LIN {X 0,Y 720.208,Z 610.953,A -85,B 0,C 180,E1 34660.965,E2 34660.965} C_VEL
LIN {X 0,Y 720.172,Z 610.956,A -85,B 0,C 180,E1 34658.142,E2 34658.142} C_VEL
LIN {X 0,Y 720.181,Z 610.956,A -85,B 0,C 180,E1 34655.418,E2 34655.418} C_VEL
LIN {X 0,Y 720.141,Z 610.957,A -85,B 0,C 180,E1 34652.468,E2 34652.468} C_VEL
LIN {X 0,Y 720.162,Z 610.958,A -85,B 0,C 180,E1 34649.922,E2 34649.922} C_VEL
LIN {X 0,Y 720.219,Z 610.948,A -85,B 0,C 180,E1 34646.977,E2 34646.977} C_VEL
LIN {X 0,Y 720.22,Z 610.957,A -85,B 0,C 180,E1 34643.945,E2 34643.945} C_VEL
LIN {X 0,Y 720.198,Z 610.951,A -85,B 0,C 180,E1 34640.975,E2 34640.975} C_VEL
LIN {X 0,Y 720.16,Z 610.957,A -85,B 0,C 180,E1 34637.899,E2 34637.899} C_VEL
LIN {X 0,Y 720.131,Z 610.96,A -85,B 0,C 180,E1 34635.403,E2 34635.403} C_VEL
LIN {X 0,Y 720.218,Z 610.954,A -85,B 0,C 180,E1 34632.551,E2 34632.551} C_VEL
LIN {X 0,Y 720.177,Z 610.955,A -85,B 0,C 180,E1 34629.692,E2 34629.692} C_VEL
LIN {X 0,Y 720.205,Z 610.955,A -85,B 0,C 180,E1 34626.953,E2 34626.953} C_VEL
LIN {X 0,Y 720.215,Z 610.951,A -85,B 0,C 180,E1 34624.069,E2 34624.069} C_VEL
LIN {X 0,Y 720.163,Z 610.958,A -85,B 0,C 180,E1 34621.2,E2 34621.2} C_VEL
LIN {X 0,Y 720.152,Z 610.959,A -85,B 0,C 180,E1 34618.625,E2 34618.625} C_VEL
LIN {X 0,Y 720.156,Z 610.958,A -85,B 0,C 180,E1 34615.556,E2 34615.556} C_VEL
LIN {X 0,Y 720.173,Z 610.957,A -85,B 0,C 180,E1 34612.948,E2 34612.948} C_VEL
LIN {X 0,Y 720.219,Z 610.95,A -85,B 0,C 180,E1 34610.002,E2 34610.002} C_VEL
LIN {X 0,Y 720.219,Z 610.959,A -85,B 0,C 180,E1 34607.02,E2 34607.02} C_VEL
LIN {X 0,Y 720.18,Z 610.954,A -85,B 0,C 180,E1 34604.13,E2 34604.13} C_VEL
LIN {X 0,Y 720.174,Z 610.961,A -85,B 0,C 180,E1 34601.152,E2 34601.152} C_VEL
LIN {X 0,Y 720.13,Z 610.962,A -85,B 0,C 180,E1 34598.564,E2 34598.564} C_VEL
LIN {X 0,Y 720.234,Z 611.091,A -85,B 0,C 180,E1 34597.759,E2 34597.759} C_VEL
LIN {X 0,Y 721.518,Z 617.349,A -85,B 0,C 180,E1 34597.269,E2 34597.269} C_VEL
LIN {X 0,Y 721.444,Z 660.306,A -85,B 0,C 180,E1 34594.24,E2 34594.24} C_VEL
LIN {X 0,Y 721.342,Z 691.441,A -85,B 0,C 180,E1 34592.016,E2 34592.016} C_VEL
LIN {X 0,Y 721.105,Z 731.111,A -85,B 0,C 180,E1 34589.212,E2 34589.212} C_VEL
LIN {X 0,Y 720.893,Z 759.497,A -85,B 0,C 180,E1 34587.193,E2 34587.193} C_VEL
LIN {X 0,Y 720.617,Z 798.923,A -85,B 0,C 180,E1 34584.386,E2 34584.386} C_VEL
LIN {X 0,Y 720.526,Z 815.5,A -85,B 0,C 180,E1 34583.249,E2 34583.249} C_VEL
LIN {X 0,Y 720.895,Z 824.532,A -85,B 0,C 180,E1 34583.152,E2 34583.152} C_VEL
LIN {X 0,Y 720.697,Z 956.974,A -85,B 0,C 180,E1 34581.81,E2 34581.81} C_VEL
LIN {X 0,Y 720.607,Z 973.104,A -85,B 0,C 180,E1 34581.493,E2 34581.493} C_VEL
LIN {X 0,Y 720.51,Z 989.356,A -85,B 0,C 180,E1 34581.02,E2 34581.02} C_VEL
LIN {X 0,Y 720.374,Z 1004.011,A -85,B 0,C 180,E1 34580.429,E2 34580.429} C_VEL
LIN {X 0,Y 720.299,Z 1015.674,A -85,B 0,C 180,E1 34579.838,E2 34579.838} C_VEL
LIN {X 0,Y 720.212,Z 1026.341,A -85,B 0,C 180,E1 34579.184,E2 34579.184} C_VEL
LIN {X 0,Y 720.127,Z 1036.599,A -85,B 0,C 180,E1 34578.427,E2 34578.427} C_VEL
LIN {X 0,Y 720.06,Z 1045.774,A -85,B 0,C 180,E1 34577.619,E2 34577.619} C_VEL
LIN {X 0,Y 719.997,Z 1054.367,A -85,B 0,C 180,E1 34576.704,E2 34576.704} C_VEL
LIN {X 0,Y 719.964,Z 1062.582,A -85,B 0,C 180,E1 34575.628,E2 34575.628} C_VEL
LIN {X 0,Y 719.931,Z 1070.175,A -85,B 0,C 180,E1 34574.311,E2 34574.311} C_VEL
LIN {X 0,Y 719.92,Z 1074.932,A -85,B 0,C 180,E1 34573.164,E2 34573.164} C_VEL
LIN {X 0,Y 719.916,Z 1077.987,A -85,B 0,C 180,E1 34572.104,E2 34572.104} C_VEL
LIN {X 0,Y 719.915,Z 1079.89,A -85,B 0,C 180,E1 34570.967,E2 34570.967} C_VEL
LIN {X 0,Y 719.916,Z 1080.431,A -85,B 0,C 180,E1 34569.834,E2 34569.834} C_VEL
LIN {X 0,Y 719.915,Z 1079.432,A -85,B 0,C 180,E1 34568.545,E2 34568.545} C_VEL
LIN {X 0,Y 719.921,Z 1076.365,A -85,B 0,C 180,E1 34567.179,E2 34567.179} C_VEL
LIN {X 0,Y 719.925,Z 1071.892,A -85,B 0,C 180,E1 34565.977,E2 34565.977} C_VEL
LIN {X 0,Y 719.942,Z 1066.603,A -85,B 0,C 180,E1 34564.938,E2 34564.938} C_VEL
LIN {X 0,Y 719.967,Z 1060.414,A -85,B 0,C 180,E1 34563.98,E2 34563.98} C_VEL
LIN {X 0,Y 720.011,Z 1052.786,A -85,B 0,C 180,E1 34563.023,E2 34563.023} C_VEL
LIN {X 0,Y 720.083,Z 1043.455,A -85,B 0,C 180,E1 34562.067,E2 34562.067} C_VEL
LIN {X 0,Y 720.187,Z 1030.252,A -85,B 0,C 180,E1 34560.993,E2 34560.993} C_VEL
LIN {X 0,Y 720.28,Z 1018.57,A -85,B 0,C 180,E1 34560.237,E2 34560.237} C_VEL
LIN {X 0,Y 720.327,Z 1007.399,A -85,B 0,C 180,E1 34559.64,E2 34559.64} C_VEL
LIN {X 0,Y 720.427,Z 995.54,A -85,B 0,C 180,E1 34559.124,E2 34559.124} C_VEL
LIN {X 0,Y 720.552,Z 982.888,A -85,B 0,C 180,E1 34558.686,E2 34558.686} C_VEL
LIN {X 0,Y 720.627,Z 969.803,A -85,B 0,C 180,E1 34558.344,E2 34558.344} C_VEL
LIN {X 0,Y 720.709,Z 954.847,A -85,B 0,C 180,E1 34558.07,E2 34558.07} C_VEL
LIN {X 0,Y 720.676,Z 816.549,A -85,B 0,C 180,E1 34556.674,E2 34556.674} C_VEL
LIN {X 0,Y 720.51,Z 814.823,A -85,B 0,C 180,E1 34556.64,E2 34556.64} C_VEL
LIN {X 0,Y 720.829,Z 771.864,A -85,B 0,C 180,E1 34553.605,E2 34553.605} C_VEL
LIN {X 0,Y 721.072,Z 739.826,A -85,B 0,C 180,E1 34551.305,E2 34551.305} C_VEL
LIN {X 0,Y 721.215,Z 704.804,A -85,B 0,C 180,E1 34548.847,E2 34548.847} C_VEL
LIN {X 0,Y 721.206,Z 667.656,A -85,B 0,C 180,E1 34546.284,E2 34546.284} C_VEL
LIN {X 0,Y 721.014,Z 625.211,A -85,B 0,C 180,E1 34543.441,E2 34543.441} C_VEL
LIN {X 0,Y 720.81,Z 613.743,A -85,B 0,C 180,E1 34542.688,E2 34542.688} C_VEL
LIN {X 0,Y 720.216,Z 610.959,A -85,B 0,C 180,E1 34542.484,E2 34542.484} C_VEL
LIN {X 0,Y 720.181,Z 610.96,A -85,B 0,C 180,E1 34539.519,E2 34539.519} C_VEL
LIN {X 0,Y 720.186,Z 610.961,A -85,B 0,C 180,E1 34536.776,E2 34536.776} C_VEL
LIN {X 0,Y 720.22,Z 610.954,A -85,B 0,C 180,E1 34533.743,E2 34533.743} C_VEL
LIN {X 0,Y 720.175,Z 610.96,A -85,B 0,C 180,E1 34530.743,E2 34530.743} C_VEL
LIN {X 0,Y 720.19,Z 610.958,A -85,B 0,C 180,E1 34527.969,E2 34527.969} C_VEL
LIN {X 0,Y 720.208,Z 610.957,A -85,B 0,C 180,E1 34524.993,E2 34524.993} C_VEL
LIN {X 0,Y 720.195,Z 610.96,A -85,B 0,C 180,E1 34522.145,E2 34522.145} C_VEL
LIN {X 0,Y 720.222,Z 610.958,A -85,B 0,C 180,E1 34519.268,E2 34519.268} C_VEL
LIN {X 0,Y 720.216,Z 610.959,A -85,B 0,C 180,E1 34516.326,E2 34516.326} C_VEL
LIN {X 0,Y 720.223,Z 610.955,A -85,B 0,C 180,E1 34513.298,E2 34513.298} C_VEL
LIN {X 0,Y 720.175,Z 610.96,A -85,B 0,C 180,E1 34510.313,E2 34510.313} C_VEL
LIN {X 0,Y 720.196,Z 610.957,A -85,B 0,C 180,E1 34507.55,E2 34507.55} C_VEL
LIN {X 0,Y 720.195,Z 610.959,A -85,B 0,C 180,E1 34504.405,E2 34504.405} C_VEL
LIN {X 0,Y 720.21,Z 611.037,A -85,B 0,C 180,E1 34502.332,E2 34502.332} C_VEL
LIN {X 0,Y 723.137,Z 620.988,A -85,B 0,C 180,E1 34501.416,E2 34501.416} C_VEL
LIN {X 0,Y 722.601,Z 658.022,A -85,B 0,C 180,E1 34498.604,E2 34498.604} C_VEL
LIN {X 0,Y 722.325,Z 683.324,A -85,B 0,C 180,E1 34496.747,E2 34496.747} C_VEL
LIN {X 0,Y 723.83,Z 691.21,A -85,B 0,C 180,E1 34496.601,E2 34496.601} C_VEL
LIN {X 0,Y 723.03,Z 975.338,A -85,B 0,C 180,E1 34493.578,E2 34493.578} C_VEL
LIN {X 0,Y 722.886,Z 996.786,A -85,B 0,C 180,E1 34493.276,E2 34493.276} C_VEL
LIN {X 0,Y 722.659,Z 1019.236,A -85,B 0,C 180,E1 34492.811,E2 34492.811} C_VEL
LIN {X 0,Y 722.426,Z 1040.16,A -85,B 0,C 180,E1 34492.234,E2 34492.234} C_VEL
LIN {X 0,Y 722.134,Z 1060.43,A -85,B 0,C 180,E1 34491.525,E2 34491.525} C_VEL
LIN {X 0,Y 721.801,Z 1080.838,A -85,B 0,C 180,E1 34490.654,E2 34490.654} C_VEL
LIN {X 0,Y 721.49,Z 1100.586,A -85,B 0,C 180,E1 34489.646,E2 34489.646} C_VEL
LIN {X 0,Y 721.179,Z 1119.415,A -85,B 0,C 180,E1 34488.51,E2 34488.51} C_VEL
LIN {X 0,Y 720.868,Z 1136.909,A -85,B 0,C 180,E1 34487.266,E2 34487.266} C_VEL
LIN {X 0,Y 720.608,Z 1152.879,A -85,B 0,C 180,E1 34485.945,E2 34485.945} C_VEL
LIN {X 0,Y 720.414,Z 1167.469,A -85,B 0,C 180,E1 34484.548,E2 34484.548} C_VEL
LIN {X 0,Y 720.248,Z 1180.679,A -85,B 0,C 180,E1 34483.077,E2 34483.077} C_VEL
LIN {X 0,Y 720.109,Z 1192.4,A -85,B 0,C 180,E1 34481.533,E2 34481.533} C_VEL
LIN {X 0,Y 720.016,Z 1203.22,A -85,B 0,C 180,E1 34479.834,E2 34479.834} C_VEL
LIN {X 0,Y 719.975,Z 1211.702,A -85,B 0,C 180,E1 34478.223,E2 34478.223} C_VEL
LIN {X 0,Y 719.924,Z 1218.675,A -85,B 0,C 180,E1 34476.538,E2 34476.538} C_VEL
LIN {X 0,Y 719.904,Z 1224.199,A -85,B 0,C 180,E1 34474.779,E2 34474.779} C_VEL
LIN {X 0,Y 719.898,Z 1227.881,A -85,B 0,C 180,E1 34473.104,E2 34473.104} C_VEL
LIN {X 0,Y 719.898,Z 1229.883,A -85,B 0,C 180,E1 34471.431,E2 34471.431} C_VEL
LIN {X 0,Y 719.898,Z 1230.396,A -85,B 0,C 180,E1 34469.601,E2 34469.601} C_VEL
LIN {X 0,Y 719.915,Z 1229.336,A -85,B 0,C 180,E1 34467.929,E2 34467.929} C_VEL
LIN {X 0,Y 719.914,Z 1226.464,A -85,B 0,C 180,E1 34466.176,E2 34466.176} C_VEL
LIN {X 0,Y 719.917,Z 1221.903,A -85,B 0,C 180,E1 34464.42,E2 34464.42} C_VEL
LIN {X 0,Y 719.946,Z 1215.93,A -85,B 0,C 180,E1 34462.738,E2 34462.738} C_VEL
LIN {X 0,Y 719.984,Z 1208.468,A -85,B 0,C 180,E1 34461.131,E2 34461.131} C_VEL
LIN {X 0,Y 720.059,Z 1198.837,A -85,B 0,C 180,E1 34459.437,E2 34459.437} C_VEL
LIN {X 0,Y 720.162,Z 1188.342,A -85,B 0,C 180,E1 34457.897,E2 34457.897} C_VEL
LIN {X 0,Y 720.305,Z 1175.652,A -85,B 0,C 180,E1 34456.339,E2 34456.339} C_VEL
LIN {X 0,Y 720.484,Z 1161.703,A -85,B 0,C 180,E1 34454.875,E2 34454.875} C_VEL
LIN {X 0,Y 720.719,Z 1146.187,A -85,B 0,C 180,E1 34453.476,E2 34453.476} C_VEL
LIN {X 0,Y 721.006,Z 1129.487,A -85,B 0,C 180,E1 34452.18,E2 34452.18} C_VEL
LIN {X 0,Y 721.309,Z 1111.316,A -85,B 0,C 180,E1 34450.981,E2 34450.981} C_VEL
LIN {X 0,Y 721.617,Z 1092.115,A -85,B 0,C 180,E1 34449.901,E2 34449.901} C_VEL
LIN {X 0,Y 721.955,Z 1071.709,A -85,B 0,C 180,E1 34448.936,E2 34448.936} C_VEL
LIN {X 0,Y 722.287,Z 1051.348,A -85,B 0,C 180,E1 34448.136,E2 34448.136} C_VEL
LIN {X 0,Y 722.517,Z 1030.436,A -85,B 0,C 180,E1 34447.48,E2 34447.48} C_VEL
LIN {X 0,Y 722.782,Z 1007.95,A -85,B 0,C 180,E1 34446.936,E2 34446.936} C_VEL
LIN {X 0,Y 722.975,Z 986.397,A -85,B 0,C 180,E1 34446.559,E2 34446.559} C_VEL
LIN {X 0,Y 723.392,Z 834.871,A -85,B 0,C 180,E1 34444.934,E2 34444.934} C_VEL
LIN {X 0,Y 723.683,Z 689.443,A -85,B 0,C 180,E1 34443.374,E2 34443.374} C_VEL
LIN {X 0,Y 722.245,Z 682.748,A -85,B 0,C 180,E1 34443.235,E2 34443.235} C_VEL
LIN {X 0,Y 722.812,Z 644.848,A -85,B 0,C 180,E1 34440.405,E2 34440.405} C_VEL
LIN {X 0,Y 723.146,Z 620.604,A -85,B 0,C 180,E1 34438.554,E2 34438.554} C_VEL
LIN {X 0,Y 720.191,Z 610.959,A -85,B 0,C 180,E1 34437.664,E2 34437.664} C_VEL
LIN {X 0,Y 720.211,Z 610.953,A -85,B 0,C 180,E1 34434.819,E2 34434.819} C_VEL
LIN {X 0,Y 720.192,Z 610.958,A -85,B 0,C 180,E1 34431.842,E2 34431.842} C_VEL
LIN {X 0,Y 720.215,Z 610.949,A -85,B 0,C 180,E1 34428.927,E2 34428.927} C_VEL
LIN {X 0,Y 720.196,Z 610.959,A -85,B 0,C 180,E1 34425.873,E2 34425.873} C_VEL
LIN {X 0,Y 720.182,Z 610.953,A -85,B 0,C 180,E1 34423.086,E2 34423.086} C_VEL
LIN {X 0,Y 720.224,Z 610.959,A -85,B 0,C 180,E1 34420.096,E2 34420.096} C_VEL
LIN {X 0,Y 720.163,Z 610.956,A -85,B 0,C 180,E1 34417.291,E2 34417.291} C_VEL
LIN {X 0,Y 720.212,Z 610.953,A -85,B 0,C 180,E1 34414.503,E2 34414.503} C_VEL
LIN {X 0,Y 720.167,Z 610.961,A -85,B 0,C 180,E1 34411.516,E2 34411.516} C_VEL
LIN {X 0,Y 720.15,Z 610.961,A -85,B 0,C 180,E1 34408.985,E2 34408.985} C_VEL
LIN {X 0,Y 720.254,Z 611.202,A -85,B 0,C 180,E1 34407.94,E2 34407.94} C_VEL
LIN {X 0,Y 721.962,Z 619.154,A -85,B 0,C 180,E1 34407.153,E2 34407.153} C_VEL
LIN {X 0,Y 722.019,Z 624.53,A -85,B 0,C 180,E1 34406.701,E2 34406.701} C_VEL
LIN {X 0,Y 723.829,Z 632.779,A -85,B 0,C 180,E1 34406.539,E2 34406.539} C_VEL
LIN {X 0,Y 723.098,Z 895.124,A -85,B 0,C 180,E1 34403.747,E2 34403.747} C_VEL
LIN {X 0,Y 722.945,Z 929.462,A -85,B 0,C 180,E1 34403.351,E2 34403.351} C_VEL
LIN {X 0,Y 722.776,Z 950.86,A -85,B 0,C 180,E1 34402.96,E2 34402.96} C_VEL
LIN {X 0,Y 722.496,Z 972.696,A -85,B 0,C 180,E1 34402.411,E2 34402.411} C_VEL
LIN {X 0,Y 722.203,Z 994.686,A -85,B 0,C 180,E1 34401.696,E2 34401.696} C_VEL
LIN {X 0,Y 721.915,Z 1015.557,A -85,B 0,C 180,E1 34400.854,E2 34400.854} C_VEL
LIN {X 0,Y 721.574,Z 1035.207,A -85,B 0,C 180,E1 34399.894,E2 34399.894} C_VEL
LIN {X 0,Y 721.25,Z 1054.058,A -85,B 0,C 180,E1 34398.805,E2 34398.805} C_VEL
LIN {X 0,Y 720.952,Z 1072.496,A -85,B 0,C 180,E1 34397.554,E2 34397.554} C_VEL
LIN {X 0,Y 720.68,Z 1089.562,A -85,B 0,C 180,E1 34396.194,E2 34396.194} C_VEL
LIN {X 0,Y 720.453,Z 1104.64,A -85,B 0,C 180,E1 34394.797,E2 34394.797} C_VEL
LIN {X 0,Y 720.257,Z 1118.345,A -85,B 0,C 180,E1 34393.305,E2 34393.305} C_VEL
LIN {X 0,Y 720.127,Z 1130.91,A -85,B 0,C 180,E1 34391.698,E2 34391.698} C_VEL
LIN {X 0,Y 720.026,Z 1141.578,A -85,B 0,C 180,E1 34390.075,E2 34390.075} C_VEL
LIN {X 0,Y 719.964,Z 1150.276,A -85,B 0,C 180,E1 34388.467,E2 34388.467} C_VEL
LIN {X 0,Y 719.924,Z 1157.686,A -85,B 0,C 180,E1 34386.757,E2 34386.757} C_VEL
LIN {X 0,Y 719.917,Z 1163.454,A -85,B 0,C 180,E1 34385.021,E2 34385.021} C_VEL
LIN {X 0,Y 719.917,Z 1167.323,A -85,B 0,C 180,E1 34383.346,E2 34383.346} C_VEL
LIN {X 0,Y 719.914,Z 1169.711,A -85,B 0,C 180,E1 34381.593,E2 34381.593} C_VEL
LIN {X 0,Y 719.91,Z 1170.475,A -85,B 0,C 180,E1 34379.843,E2 34379.843} C_VEL
LIN {X 0,Y 719.911,Z 1169.52,A -85,B 0,C 180,E1 34378.092,E2 34378.092} C_VEL
LIN {X 0,Y 719.915,Z 1166.879,A -85,B 0,C 180,E1 34376.339,E2 34376.339} C_VEL
LIN {X 0,Y 719.926,Z 1162.567,A -85,B 0,C 180,E1 34374.583,E2 34374.583} C_VEL
LIN {X 0,Y 719.942,Z 1156.731,A -85,B 0,C 180,E1 34372.902,E2 34372.902} C_VEL
LIN {X 0,Y 719.976,Z 1149.125,A -85,B 0,C 180,E1 34371.215,E2 34371.215} C_VEL
LIN {X 0,Y 720.041,Z 1140.185,A -85,B 0,C 180,E1 34369.602,E2 34369.602} C_VEL
LIN {X 0,Y 720.135,Z 1129.841,A -85,B 0,C 180,E1 34368.062,E2 34368.062} C_VEL
LIN {X 0,Y 720.269,Z 1117.57,A -85,B 0,C 180,E1 34366.515,E2 34366.515} C_VEL
LIN {X 0,Y 720.461,Z 1103.912,A -85,B 0,C 180,E1 34365.042,E2 34365.042} C_VEL
LIN {X 0,Y 720.489,Z 1101.611,A -85,B 0,C 180,E1 34364.82,E2 34364.82} C_VEL
LIN {X 0,Y 719.582,Z 1096.843,A -85,B 0,C 180,E1 34364.341,E2 34364.341} C_VEL
LIN {X 0,Y 713.69,Z 1083.945,A -85,B 0,C 180,E1 34363.074,E2 34363.074} C_VEL
LIN {X 0,Y 713.042,Z 1079.38,A -85,B 0,C 180,E1 34362.686,E2 34362.686} C_VEL
LIN {X 0,Y 713.399,Z 1061.921,A -85,B 0,C 180,E1 34361.408,E2 34361.408} C_VEL
LIN {X 0,Y 713.782,Z 1043.036,A -85,B 0,C 180,E1 34360.229,E2 34360.229} C_VEL
LIN {X 0,Y 714.179,Z 1022.968,A -85,B 0,C 180,E1 34359.171,E2 34359.171} C_VEL
LIN {X 0,Y 714.582,Z 1002.755,A -85,B 0,C 180,E1 34358.28,E2 34358.28} C_VEL
LIN {X 0,Y 714.928,Z 981.908,A -85,B 0,C 180,E1 34357.534,E2 34357.534} C_VEL
LIN {X 0,Y 715.253,Z 959.699,A -85,B 0,C 180,E1 34356.905,E2 34356.905} C_VEL
LIN {X 0,Y 715.521,Z 937.487,A -85,B 0,C 180,E1 34356.436,E2 34356.436} C_VEL
LIN {X 0,Y 715.69,Z 915.823,A -85,B 0,C 180,E1 34356.126,E2 34356.126} C_VEL
LIN {X 0,Y 716.689,Z 640.954,A -85,B 0,C 180,E1 34353.175,E2 34353.175} C_VEL
LIN {X 0,Y 716.479,Z 632.558,A -85,B 0,C 180,E1 34353.074,E2 34353.074} C_VEL
LIN {X 0,Y 714.354,Z 623.95,A -85,B 0,C 180,E1 34352.878,E2 34352.878} C_VEL
LIN {X 0,Y 714.269,Z 619.697,A -85,B 0,C 180,E1 34352.489,E2 34352.489} C_VEL
LIN {X 0,Y 712.232,Z 611.949,A -85,B 0,C 180,E1 34351.671,E2 34351.671} C_VEL
LIN {X 0,Y 712.231,Z 611.95,A -85,B 0,C 180,E1 34348.99,E2 34348.99} C_VEL
LIN {X 0,Y 712.204,Z 611.949,A -85,B 0,C 180,E1 34345.935,E2 34345.935} C_VEL
LIN {X 0,Y 712.231,Z 611.948,A -85,B 0,C 180,E1 34343.373,E2 34343.373} C_VEL
LIN {X 0,Y 712.281,Z 611.938,A -85,B 0,C 180,E1 34340.411,E2 34340.411} C_VEL
LIN {X 0,Y 712.276,Z 611.948,A -85,B 0,C 180,E1 34337.358,E2 34337.358} C_VEL
LIN {X 0,Y 712.268,Z 611.94,A -85,B 0,C 180,E1 34334.355,E2 34334.355} C_VEL
LIN {X 0,Y 712.218,Z 611.949,A -85,B 0,C 180,E1 34331.395,E2 34331.395} C_VEL
LIN {X 0,Y 712.197,Z 611.949,A -85,B 0,C 180,E1 34328.871,E2 34328.871} C_VEL
LIN {X 0,Y 712.271,Z 611.942,A -85,B 0,C 180,E1 34325.909,E2 34325.909} C_VEL
LIN {X 0,Y 712.249,Z 611.946,A -85,B 0,C 180,E1 34323.004,E2 34323.004} C_VEL
LIN {X 0,Y 712.267,Z 611.939,A -85,B 0,C 180,E1 34320.078,E2 34320.078} C_VEL
LIN {X 0,Y 712.274,Z 611.948,A -85,B 0,C 180,E1 34317.055,E2 34317.055} C_VEL
LIN {X 0,Y 712.218,Z 611.946,A -85,B 0,C 180,E1 34314.29,E2 34314.29} C_VEL
LIN {X 0,Y 712.253,Z 611.949,A -85,B 0,C 180,E1 34311.408,E2 34311.408} C_VEL
LIN {X 0,Y 712.208,Z 611.946,A -85,B 0,C 180,E1 34308.67,E2 34308.67} C_VEL
LIN {X 0,Y 712.28,Z 611.946,A -85,B 0,C 180,E1 34305.888,E2 34305.888} C_VEL
LIN {X 0,Y 712.26,Z 611.939,A -85,B 0,C 180,E1 34302.981,E2 34302.981} C_VEL
LIN {X 0,Y 712.251,Z 611.944,A -85,B 0,C 180,E1 34300.108,E2 34300.108} C_VEL
LIN {X 0,Y 712.28,Z 611.94,A -85,B 0,C 180,E1 34297.178,E2 34297.178} C_VEL
LIN {X 0,Y 712.2,Z 611.948,A -85,B 0,C 180,E1 34294.349,E2 34294.349} C_VEL
LIN {X 0,Y 712.214,Z 611.946,A -85,B 0,C 180,E1 34291.743,E2 34291.743} C_VEL
LIN {X 0,Y 712.247,Z 611.942,A -85,B 0,C 180,E1 34288.634,E2 34288.634} C_VEL
LIN {X 0,Y 712.278,Z 611.945,A -85,B 0,C 180,E1 34285.734,E2 34285.734} C_VEL
LIN {X 0,Y 712.281,Z 611.938,A -85,B 0,C 180,E1 34282.743,E2 34282.743} C_VEL
LIN {X 0,Y 712.234,Z 611.944,A -85,B 0,C 180,E1 34279.758,E2 34279.758} C_VEL
LIN {X 0,Y 712.219,Z 611.945,A -85,B 0,C 180,E1 34277.103,E2 34277.103} C_VEL
LIN {X 0,Y 712.212,Z 611.947,A -85,B 0,C 180,E1 34274.029,E2 34274.029} C_VEL
LIN {X 0,Y 712.23,Z 611.946,A -85,B 0,C 180,E1 34271.418,E2 34271.418} C_VEL
LIN {X 0,Y 712.283,Z 611.938,A -85,B 0,C 180,E1 34268.422,E2 34268.422} C_VEL
LIN {X 0,Y 712.277,Z 611.948,A -85,B 0,C 180,E1 34265.361,E2 34265.361} C_VEL
LIN {X 0,Y 712.262,Z 611.941,A -85,B 0,C 180,E1 34262.404,E2 34262.404} C_VEL
LIN {X 0,Y 712.213,Z 611.948,A -85,B 0,C 180,E1 34259.379,E2 34259.379} C_VEL
LIN {X 0,Y 712.195,Z 611.949,A -85,B 0,C 180,E1 34256.899,E2 34256.899} C_VEL
LIN {X 0,Y 712.276,Z 611.942,A -85,B 0,C 180,E1 34253.953,E2 34253.953} C_VEL
LIN {X 0,Y 712.249,Z 611.946,A -85,B 0,C 180,E1 34251.031,E2 34251.031} C_VEL
LIN {X 0,Y 712.263,Z 611.941,A -85,B 0,C 180,E1 34248.181,E2 34248.181} C_VEL
LIN {X 0,Y 712.279,Z 611.947,A -85,B 0,C 180,E1 34245.143,E2 34245.143} C_VEL
LIN {X 0,Y 712.215,Z 611.947,A -85,B 0,C 180,E1 34242.364,E2 34242.364} C_VEL
LIN {X 0,Y 712.263,Z 611.949,A -85,B 0,C 180,E1 34239.486,E2 34239.486} C_VEL
LIN {X 0,Y 712.27,Z 612.124,A -85,B 0,C 180,E1 34237.952,E2 34237.952} C_VEL
LIN {X 0,Y 713.889,Z 619.31,A -85,B 0,C 180,E1 34237.387,E2 34237.387} C_VEL
LIN {X 0,Y 713.757,Z 663.317,A -85,B 0,C 180,E1 34234.26,E2 34234.26} C_VEL
LIN {X 0,Y 713.591,Z 701.946,A -85,B 0,C 180,E1 34231.507,E2 34231.507} C_VEL
LIN {X 0,Y 713.355,Z 742.215,A -85,B 0,C 180,E1 34228.642,E2 34228.642} C_VEL
LIN {X 0,Y 713.008,Z 777.238,A -85,B 0,C 180,E1 34226.123,E2 34226.123} C_VEL
LIN {X 0,Y 712.643,Z 815.347,A -85,B 0,C 180,E1 34223.401,E2 34223.401} C_VEL
LIN {X 0,Y 713.107,Z 823.548,A -85,B 0,C 180,E1 34223.309,E2 34223.309} C_VEL
LIN {X 0,Y 712.864,Z 956.883,A -85,B 0,C 180,E1 34221.943,E2 34221.943} C_VEL
LIN {X 0,Y 712.761,Z 972.125,A -85,B 0,C 180,E1 34221.643,E2 34221.643} C_VEL
LIN {X 0,Y 712.665,Z 987.139,A -85,B 0,C 180,E1 34221.22,E2 34221.22} C_VEL
LIN {X 0,Y 712.497,Z 1002.672,A -85,B 0,C 180,E1 34220.609,E2 34220.609} C_VEL
LIN {X 0,Y 712.392,Z 1015.074,A -85,B 0,C 180,E1 34219.982,E2 34219.982} C_VEL
LIN {X 0,Y 712.283,Z 1026.015,A -85,B 0,C 180,E1 34219.309,E2 34219.309} C_VEL
LIN {X 0,Y 712.183,Z 1035.86,A -85,B 0,C 180,E1 34218.582,E2 34218.582} C_VEL
LIN {X 0,Y 712.107,Z 1044.552,A -85,B 0,C 180,E1 34217.822,E2 34217.822} C_VEL
LIN {X 0,Y 712.035,Z 1052.626,A -85,B 0,C 180,E1 34216.981,E2 34216.981} C_VEL
LIN {X 0,Y 711.984,Z 1059.961,A -85,B 0,C 180,E1 34216.059,E2 34216.059} C_VEL
LIN {X 0,Y 711.951,Z 1065.949,A -85,B 0,C 180,E1 34215.141,E2 34215.141} C_VEL
LIN {X 0,Y 711.933,Z 1071.139,A -85,B 0,C 180,E1 34214.143,E2 34214.143} C_VEL
LIN {X 0,Y 711.92,Z 1075.087,A -85,B 0,C 180,E1 34213.15,E2 34213.15} C_VEL
LIN {X 0,Y 711.916,Z 1078.084,A -85,B 0,C 180,E1 34212.078,E2 34212.078} C_VEL
LIN {X 0,Y 711.916,Z 1079.881,A -85,B 0,C 180,E1 34210.974,E2 34210.974} C_VEL
LIN {X 0,Y 711.917,Z 1080.416,A -85,B 0,C 180,E1 34209.864,E2 34209.864} C_VEL
LIN {X 0,Y 711.915,Z 1079.531,A -85,B 0,C 180,E1 34208.608,E2 34208.608} C_VEL
LIN {X 0,Y 711.921,Z 1076.459,A -85,B 0,C 180,E1 34207.179,E2 34207.179} C_VEL
LIN {X 0,Y 711.928,Z 1072.379,A -85,B 0,C 180,E1 34206.045,E2 34206.045} C_VEL
LIN {X 0,Y 711.947,Z 1067.231,A -85,B 0,C 180,E1 34204.994,E2 34204.994} C_VEL
LIN {X 0,Y 711.976,Z 1061.192,A -85,B 0,C 180,E1 34204.025,E2 34204.025} C_VEL
LIN {X 0,Y 712.017,Z 1054.418,A -85,B 0,C 180,E1 34203.138,E2 34203.138} C_VEL
LIN {X 0,Y 712.088,Z 1046.234,A -85,B 0,C 180,E1 34202.251,E2 34202.251} C_VEL
LIN {X 0,Y 712.17,Z 1037.305,A -85,B 0,C 180,E1 34201.446,E2 34201.446} C_VEL
LIN {X 0,Y 712.264,Z 1027.776,A -85,B 0,C 180,E1 34200.722,E2 34200.722} C_VEL
LIN {X 0,Y 712.364,Z 1017.697,A -85,B 0,C 180,E1 34200.079,E2 34200.079} C_VEL
LIN {X 0,Y 712.429,Z 1007.182,A -85,B 0,C 180,E1 34199.516,E2 34199.516} C_VEL
LIN {X 0,Y 712.551,Z 995.271,A -85,B 0,C 180,E1 34198.993,E2 34198.993} C_VEL
LIN {X 0,Y 712.682,Z 983.862,A -85,B 0,C 180,E1 34198.591,E2 34198.591} C_VEL
LIN {X 0,Y 712.773,Z 971.223,A -85,B 0,C 180,E1 34198.247,E2 34198.247} C_VEL
LIN {X 0,Y 712.865,Z 956.628,A -85,B 0,C 180,E1 34197.964,E2 34197.964} C_VEL
LIN {X 0,Y 712.889,Z 817.239,A -85,B 0,C 180,E1 34196.533,E2 34196.533} C_VEL
LIN {X 0,Y 712.643,Z 814.973,A -85,B 0,C 180,E1 34196.499,E2 34196.499} C_VEL
LIN {X 0,Y 713.106,Z 772.038,A -85,B 0,C 180,E1 34193.396,E2 34193.396} C_VEL
LIN {X 0,Y 713.336,Z 745.498,A -85,B 0,C 180,E1 34191.494,E2 34191.494} C_VEL
LIN {X 0,Y 713.461,Z 706.642,A -85,B 0,C 180,E1 34188.765,E2 34188.765} C_VEL
LIN {X 0,Y 713.475,Z 670.947,A -85,B 0,C 180,E1 34186.298,E2 34186.298} C_VEL
LIN {X 0,Y 713.258,Z 630.642,A -85,B 0,C 180,E1 34183.591,E2 34183.591} C_VEL
LIN {X 0,Y 713.019,Z 615.291,A -85,B 0,C 180,E1 34182.577,E2 34182.577} C_VEL
LIN {X 0,Y 712.275,Z 611.947,A -85,B 0,C 180,E1 34182.326,E2 34182.326} C_VEL
LIN {X 0,Y 712.234,Z 611.949,A -85,B 0,C 180,E1 34179.28,E2 34179.28} C_VEL
LIN {X 0,Y 712.241,Z 611.95,A -85,B 0,C 180,E1 34176.59,E2 34176.59} C_VEL
LIN {X 0,Y 712.273,Z 611.945,A -85,B 0,C 180,E1 34173.485,E2 34173.485} C_VEL
LIN {X 0,Y 712.246,Z 611.949,A -85,B 0,C 180,E1 34170.569,E2 34170.569} C_VEL
LIN {X 0,Y 712.276,Z 611.946,A -85,B 0,C 180,E1 34167.665,E2 34167.665} C_VEL
LIN {X 0,Y 712.28,Z 611.948,A -85,B 0,C 180,E1 34164.644,E2 34164.644} C_VEL
LIN {X 0,Y 712.283,Z 611.944,A -85,B 0,C 180,E1 34161.562,E2 34161.562} C_VEL
LIN {X 0,Y 712.234,Z 611.948,A -85,B 0,C 180,E1 34158.498,E2 34158.498} C_VEL
LIN {X 0,Y 712.255,Z 611.946,A -85,B 0,C 180,E1 34155.719,E2 34155.719} C_VEL
LIN {X 0,Y 712.262,Z 611.945,A -85,B 0,C 180,E1 34152.641,E2 34152.641} C_VEL
LIN {X 0,Y 712.246,Z 611.949,A -85,B 0,C 180,E1 34149.801,E2 34149.801} C_VEL
LIN {X 0,Y 712.285,Z 611.946,A -85,B 0,C 180,E1 34146.826,E2 34146.826} C_VEL
LIN {X 0,Y 712.279,Z 611.949,A -85,B 0,C 180,E1 34143.868,E2 34143.868} C_VEL
LIN {X 0,Y 712.318,Z 612.184,A -85,B 0,C 180,E1 34142.623,E2 34142.623} C_VEL
LIN {X 0,Y 715.782,Z 623.742,A -85,B 0,C 180,E1 34141.556,E2 34141.556} C_VEL
LIN {X 0,Y 715.155,Z 660.411,A -85,B 0,C 180,E1 34138.746,E2 34138.746} C_VEL
LIN {X 0,Y 714.859,Z 683.329,A -85,B 0,C 180,E1 34137.049,E2 34137.049} C_VEL
LIN {X 0,Y 716.67,Z 692.713,A -85,B 0,C 180,E1 34136.872,E2 34136.872} C_VEL
LIN {X 0,Y 715.685,Z 976.194,A -85,B 0,C 180,E1 34133.824,E2 34133.824} C_VEL
LIN {X 0,Y 715.519,Z 997.499,A -85,B 0,C 180,E1 34133.518,E2 34133.518} C_VEL
LIN {X 0,Y 715.246,Z 1019.57,A -85,B 0,C 180,E1 34133.053,E2 34133.053} C_VEL
LIN {X 0,Y 714.973,Z 1039.924,A -85,B 0,C 180,E1 34132.486,E2 34132.486} C_VEL
LIN {X 0,Y 714.612,Z 1060.434,A -85,B 0,C 180,E1 34131.763,E2 34131.763} C_VEL
LIN {X 0,Y 714.215,Z 1081.097,A -85,B 0,C 180,E1 34130.871,E2 34130.871} C_VEL
LIN {X 0,Y 713.833,Z 1100.745,A -85,B 0,C 180,E1 34129.856,E2 34129.856} C_VEL
LIN {X 0,Y 713.454,Z 1119.415,A -85,B 0,C 180,E1 34128.718,E2 34128.718} C_VEL
LIN {X 0,Y 713.081,Z 1136.91,A -85,B 0,C 180,E1 34127.461,E2 34127.461} C_VEL
LIN {X 0,Y 712.772,Z 1152.879,A -85,B 0,C 180,E1 34126.125,E2 34126.125} C_VEL
LIN {X 0,Y 712.529,Z 1167.47,A -85,B 0,C 180,E1 34124.713,E2 34124.713} C_VEL
LIN {X 0,Y 712.319,Z 1180.678,A -85,B 0,C 180,E1 34123.225,E2 34123.225} C_VEL
LIN {X 0,Y 712.151,Z 1192.401,A -85,B 0,C 180,E1 34121.663,E2 34121.663} C_VEL
LIN {X 0,Y 712.042,Z 1203.22,A -85,B 0,C 180,E1 34119.945,E2 34119.945} C_VEL
LIN {X 0,Y 711.989,Z 1211.702,A -85,B 0,C 180,E1 34118.316,E2 34118.316} C_VEL
LIN {X 0,Y 711.926,Z 1218.675,A -85,B 0,C 180,E1 34116.612,E2 34116.612} C_VEL
LIN {X 0,Y 711.904,Z 1224.2,A -85,B 0,C 180,E1 34114.833,E2 34114.833} C_VEL
LIN {X 0,Y 711.9,Z 1227.881,A -85,B 0,C 180,E1 34113.139,E2 34113.139} C_VEL
LIN {X 0,Y 711.899,Z 1229.884,A -85,B 0,C 180,E1 34111.448,E2 34111.448} C_VEL
LIN {X 0,Y 711.898,Z 1230.396,A -85,B 0,C 180,E1 34109.597,E2 34109.597} C_VEL
LIN {X 0,Y 711.915,Z 1229.336,A -85,B 0,C 180,E1 34107.906,E2 34107.906} C_VEL
LIN {X 0,Y 711.915,Z 1226.463,A -85,B 0,C 180,E1 34106.133,E2 34106.133} C_VEL
LIN {X 0,Y 711.917,Z 1221.903,A -85,B 0,C 180,E1 34104.357,E2 34104.357} C_VEL
LIN {X 0,Y 711.95,Z 1215.93,A -85,B 0,C 180,E1 34102.656,E2 34102.656} C_VEL
LIN {X 0,Y 712,Z 1208.468,A -85,B 0,C 180,E1 34101.031,E2 34101.031} C_VEL
LIN {X 0,Y 712.086,Z 1198.836,A -85,B 0,C 180,E1 34099.317,E2 34099.317} C_VEL
LIN {X 0,Y 712.225,Z 1188.044,A -85,B 0,C 180,E1 34097.72,E2 34097.72} C_VEL
LIN {X 0,Y 712.393,Z 1175.739,A -85,B 0,C 180,E1 34096.195,E2 34096.195} C_VEL
LIN {X 0,Y 712.615,Z 1161.703,A -85,B 0,C 180,E1 34094.704,E2 34094.704} C_VEL
LIN {X 0,Y 712.891,Z 1146.683,A -85,B 0,C 180,E1 34093.33,E2 34093.33} C_VEL
LIN {X 0,Y 713.23,Z 1130.236,A -85,B 0,C 180,E1 34092.035,E2 34092.035} C_VEL
LIN {X 0,Y 713.582,Z 1112.76,A -85,B 0,C 180,E1 34090.859,E2 34090.859} C_VEL
LIN {X 0,Y 713.979,Z 1092.92,A -85,B 0,C 180,E1 34089.719,E2 34089.719} C_VEL
LIN {X 0,Y 714.378,Z 1073.484,A -85,B 0,C 180,E1 34088.778,E2 34088.778} C_VEL
LIN {X 0,Y 714.742,Z 1053.616,A -85,B 0,C 180,E1 34087.98,E2 34087.98} C_VEL
LIN {X 0,Y 715.049,Z 1032.653,A -85,B 0,C 180,E1 34087.297,E2 34087.297} C_VEL
LIN {X 0,Y 715.38,Z 1010.918,A -85,B 0,C 180,E1 34086.745,E2 34086.745} C_VEL
LIN {X 0,Y 715.577,Z 989.77,A -85,B 0,C 180,E1 34086.354,E2 34086.354} C_VEL
LIN {X 0,Y 715.772,Z 956.487,A -85,B 0,C 180,E1 34085.964,E2 34085.964} C_VEL
LIN {X 0,Y 716.63,Z 691.362,A -85,B 0,C 180,E1 34083.112,E2 34083.112} C_VEL
LIN {X 0,Y 714.779,Z 682.778,A -85,B 0,C 180,E1 34082.935,E2 34082.935} C_VEL
LIN {X 0,Y 715.458,Z 643.653,A -85,B 0,C 180,E1 34079.978,E2 34079.978} C_VEL
LIN {X 0,Y 715.71,Z 623.186,A -85,B 0,C 180,E1 34078.405,E2 34078.405} C_VEL
LIN {X 0,Y 712.259,Z 611.946,A -85,B 0,C 180,E1 34077.403,E2 34077.403} C_VEL
LIN {X 0,Y 712.271,Z 611.948,A -85,B 0,C 180,E1 34074.466,E2 34074.466} C_VEL
LIN {X 0,Y 712.244,Z 611.945,A -85,B 0,C 180,E1 34071.57,E2 34071.57} C_VEL
LIN {X 0,Y 712.277,Z 611.941,A -85,B 0,C 180,E1 34068.681,E2 34068.681} C_VEL
LIN {X 0,Y 712.245,Z 611.947,A -85,B 0,C 180,E1 34065.724,E2 34065.724} C_VEL
LIN {X 0,Y 712.261,Z 611.941,A -85,B 0,C 180,E1 34062.878,E2 34062.878} C_VEL
LIN {X 0,Y 712.252,Z 611.949,A -85,B 0,C 180,E1 34059.804,E2 34059.804} C_VEL
LIN {X 0,Y 712.227,Z 611.945,A -85,B 0,C 180,E1 34057.116,E2 34057.116} C_VEL
LIN {X 0,Y 712.282,Z 611.946,A -85,B 0,C 180,E1 34054.225,E2 34054.225} C_VEL
LIN {X 0,Y 712.22,Z 611.949,A -85,B 0,C 180,E1 34051.39,E2 34051.39} C_VEL
LIN {X 0,Y 712.222,Z 611.95,A -85,B 0,C 180,E1 34048.787,E2 34048.787} C_VEL
LIN {X 0,Y 712.285,Z 611.955,A -85,B 0,C 180,E1 34048.212,E2 34048.212} C_VEL
LIN {X 0,Y 714.389,Z 621.646,A -85,B 0,C 180,E1 34047.239,E2 34047.239} C_VEL
LIN {X 0,Y 714.465,Z 624.558,A -85,B 0,C 180,E1 34047.006,E2 34047.006} C_VEL
LIN {X 0,Y 716.665,Z 634.327,A -85,B 0,C 180,E1 34046.809,E2 34046.809} C_VEL
LIN {X 0,Y 715.771,Z 896.635,A -85,B 0,C 180,E1 34043.989,E2 34043.989} C_VEL
LIN {X 0,Y 715.591,Z 929.654,A -85,B 0,C 180,E1 34043.603,E2 34043.603} C_VEL
LIN {X 0,Y 715.386,Z 951.094,A -85,B 0,C 180,E1 34043.207,E2 34043.207} C_VEL
LIN {X 0,Y 715.059,Z 972.156,A -85,B 0,C 180,E1 34042.673,E2 34042.673} C_VEL
LIN {X 0,Y 714.735,Z 993.548,A -85,B 0,C 180,E1 34041.978,E2 34041.978} C_VEL
LIN {X 0,Y 714.38,Z 1013.672,A -85,B 0,C 180,E1 34041.17,E2 34041.17} C_VEL
LIN {X 0,Y 713.963,Z 1033.697,A -85,B 0,C 180,E1 34040.197,E2 34040.197} C_VEL
LIN {X 0,Y 713.571,Z 1053.411,A -85,B 0,C 180,E1 34039.057,E2 34039.057} C_VEL
LIN {X 0,Y 713.194,Z 1071.868,A -85,B 0,C 180,E1 34037.798,E2 34037.798} C_VEL
LIN {X 0,Y 712.868,Z 1088.615,A -85,B 0,C 180,E1 34036.461,E2 34036.461} C_VEL
LIN {X 0,Y 712.587,Z 1103.803,A -85,B 0,C 180,E1 34035.047,E2 34035.047} C_VEL
LIN {X 0,Y 712.356,Z 1117.475,A -85,B 0,C 180,E1 34033.558,E2 34033.558} C_VEL
LIN {X 0,Y 712.189,Z 1130.339,A -85,B 0,C 180,E1 34031.912,E2 34031.912} C_VEL
LIN {X 0,Y 712.061,Z 1141.089,A -85,B 0,C 180,E1 34030.274,E2 34030.274} C_VEL
LIN {X 0,Y 711.982,Z 1149.953,A -85,B 0,C 180,E1 34028.628,E2 34028.628} C_VEL
LIN {X 0,Y 711.931,Z 1157.599,A -85,B 0,C 180,E1 34026.858,E2 34026.858} C_VEL
LIN {X 0,Y 711.926,Z 1163.244,A -85,B 0,C 180,E1 34025.159,E2 34025.159} C_VEL
LIN {X 0,Y 711.917,Z 1167.168,A -85,B 0,C 180,E1 34023.464,E2 34023.464} C_VEL
LIN {X 0,Y 711.914,Z 1169.712,A -85,B 0,C 180,E1 34021.611,E2 34021.611} C_VEL
LIN {X 0,Y 711.91,Z 1170.475,A -85,B 0,C 180,E1 34019.841,E2 34019.841} C_VEL
LIN {X 0,Y 711.913,Z 1169.588,A -85,B 0,C 180,E1 34018.151,E2 34018.151} C_VEL
LIN {X 0,Y 711.916,Z 1167.037,A -85,B 0,C 180,E1 34016.378,E2 34016.378} C_VEL
LIN {X 0,Y 711.928,Z 1162.82,A -85,B 0,C 180,E1 34014.602,E2 34014.602} C_VEL
LIN {X 0,Y 711.947,Z 1157.036,A -85,B 0,C 180,E1 34012.903,E2 34012.903} C_VEL
LIN {X 0,Y 711.999,Z 1149.124,A -85,B 0,C 180,E1 34011.115,E2 34011.115} C_VEL
LIN {X 0,Y 712.077,Z 1140.184,A -85,B 0,C 180,E1 34009.484,E2 34009.484} C_VEL
LIN {X 0,Y 712.19,Z 1129.835,A -85,B 0,C 180,E1 34007.927,E2 34007.927} C_VEL
LIN {X 0,Y 712.372,Z 1116.863,A -85,B 0,C 180,E1 34006.28,E2 34006.28} C_VEL
LIN {X 0,Y 712.606,Z 1102.613,A -85,B 0,C 180,E1 34004.746,E2 34004.746} C_VEL
LIN {X 0,Y 712.888,Z 1087.247,A -85,B 0,C 180,E1 34003.33,E2 34003.33} C_VEL
LIN {X 0,Y 713.042,Z 1079.38,A -85,B 0,C 180,E1 34002.686,E2 34002.686} C_VEL
LIN {X 0,Y 712.178,Z 1074.006,A -85,B 0,C 180,E1 34002.24,E2 34002.24} C_VEL
LIN {X 0,Y 706.657,Z 1060.469,A -85,B 0,C 180,E1 34001.122,E2 34001.122} C_VEL
LIN {X 0,Y 705.853,Z 1054.615,A -85,B 0,C 180,E1 34000.713,E2 34000.713} C_VEL
LIN {X 0,Y 706.31,Z 1035.493,A -85,B 0,C 180,E1 33999.581,E2 33999.581} C_VEL
LIN {X 0,Y 706.785,Z 1015.703,A -85,B 0,C 180,E1 33998.595,E2 33998.595} C_VEL
LIN {X 0,Y 707.203,Z 995.552,A -85,B 0,C 180,E1 33997.762,E2 33997.762} C_VEL
LIN {X 0,Y 707.62,Z 973.57,A -85,B 0,C 180,E1 33997.026,E2 33997.026} C_VEL
LIN {X 0,Y 708.001,Z 951.788,A -85,B 0,C 180,E1 33996.461,E2 33996.461} C_VEL
LIN {X 0,Y 708.234,Z 930.159,A -85,B 0,C 180,E1 33996.055,E2 33996.055} C_VEL
LIN {X 0,Y 708.453,Z 898.268,A -85,B 0,C 180,E1 33995.674,E2 33995.674} C_VEL
LIN {X 0,Y 709.535,Z 634.886,A -85,B 0,C 180,E1 33992.815,E2 33992.815} C_VEL
LIN {X 0,Y 706.806,Z 623.919,A -85,B 0,C 180,E1 33992.562,E2 33992.562} C_VEL
LIN {X 0,Y 706.065,Z 619.69,A -85,B 0,C 180,E1 33992.142,E2 33992.142} C_VEL
LIN {X 0,Y 704.287,Z 612.938,A -85,B 0,C 180,E1 33991.419,E2 33991.419} C_VEL
LIN {X 0,Y 704.341,Z 612.938,A -85,B 0,C 180,E1 33988.508,E2 33988.508} C_VEL
LIN {X 0,Y 704.258,Z 612.939,A -85,B 0,C 180,E1 33985.694,E2 33985.694} C_VEL
LIN {X 0,Y 704.333,Z 612.937,A -85,B 0,C 180,E1 33982.995,E2 33982.995} C_VEL
LIN {X 0,Y 704.314,Z 612.93,A -85,B 0,C 180,E1 33979.979,E2 33979.979} C_VEL
LIN {X 0,Y 704.321,Z 612.934,A -85,B 0,C 180,E1 33977.1,E2 33977.1} C_VEL
LIN {X 0,Y 704.345,Z 612.929,A -85,B 0,C 180,E1 33974.189,E2 33974.189} C_VEL
LIN {X 0,Y 704.273,Z 612.937,A -85,B 0,C 180,E1 33971.314,E2 33971.314} C_VEL
LIN {X 0,Y 704.264,Z 612.938,A -85,B 0,C 180,E1 33968.765,E2 33968.765} C_VEL
LIN {X 0,Y 704.307,Z 612.931,A -85,B 0,C 180,E1 33965.697,E2 33965.697} C_VEL
LIN {X 0,Y 704.325,Z 612.936,A -85,B 0,C 180,E1 33962.82,E2 33962.82} C_VEL
LIN {X 0,Y 704.342,Z 612.926,A -85,B 0,C 180,E1 33959.793,E2 33959.793} C_VEL
LIN {X 0,Y 704.307,Z 612.934,A -85,B 0,C 180,E1 33956.747,E2 33956.747} C_VEL
LIN {X 0,Y 704.305,Z 612.934,A -85,B 0,C 180,E1 33953.956,E2 33953.956} C_VEL
LIN {X 0,Y 704.259,Z 612.938,A -85,B 0,C 180,E1 33950.907,E2 33950.907} C_VEL
LIN {X 0,Y 704.282,Z 612.936,A -85,B 0,C 180,E1 33948.373,E2 33948.373} C_VEL
LIN {X 0,Y 704.342,Z 612.927,A -85,B 0,C 180,E1 33945.396,E2 33945.396} C_VEL
LIN {X 0,Y 704.338,Z 612.935,A -85,B 0,C 180,E1 33942.379,E2 33942.379} C_VEL
LIN {X 0,Y 704.338,Z 612.927,A -85,B 0,C 180,E1 33939.314,E2 33939.314} C_VEL
LIN {X 0,Y 704.286,Z 612.937,A -85,B 0,C 180,E1 33936.359,E2 33936.359} C_VEL
LIN {X 0,Y 704.256,Z 612.937,A -85,B 0,C 180,E1 33933.827,E2 33933.827} C_VEL
LIN {X 0,Y 704.313,Z 612.933,A -85,B 0,C 180,E1 33930.815,E2 33930.815} C_VEL
LIN {X 0,Y 704.299,Z 612.934,A -85,B 0,C 180,E1 33928.035,E2 33928.035} C_VEL
LIN {X 0,Y 704.332,Z 612.927,A -85,B 0,C 180,E1 33925.115,E2 33925.115} C_VEL
LIN {X 0,Y 704.343,Z 612.936,A -85,B 0,C 180,E1 33922.086,E2 33922.086} C_VEL
LIN {X 0,Y 704.29,Z 612.93,A -85,B 0,C 180,E1 33919.231,E2 33919.231} C_VEL
LIN {X 0,Y 704.305,Z 612.937,A -85,B 0,C 180,E1 33916.287,E2 33916.287} C_VEL
LIN {X 0,Y 704.261,Z 612.936,A -85,B 0,C 180,E1 33913.59,E2 33913.59} C_VEL
LIN {X 0,Y 704.344,Z 612.933,A -85,B 0,C 180,E1 33910.772,E2 33910.772} C_VEL
LIN {X 0,Y 704.313,Z 612.932,A -85,B 0,C 180,E1 33907.815,E2 33907.815} C_VEL
LIN {X 0,Y 704.315,Z 612.932,A -85,B 0,C 180,E1 33904.974,E2 33904.974} C_VEL
LIN {X 0,Y 704.344,Z 612.932,A -85,B 0,C 180,E1 33902,E2 33902} C_VEL
LIN {X 0,Y 704.262,Z 612.937,A -85,B 0,C 180,E1 33899.169,E2 33899.169} C_VEL
LIN {X 0,Y 704.296,Z 612.938,A -85,B 0,C 180,E1 33896.48,E2 33896.48} C_VEL
LIN {X 0,Y 704.291,Z 612.933,A -85,B 0,C 180,E1 33893.466,E2 33893.466} C_VEL
LIN {X 0,Y 704.34,Z 612.937,A -85,B 0,C 180,E1 33890.614,E2 33890.614} C_VEL
LIN {X 0,Y 704.332,Z 612.929,A -85,B 0,C 180,E1 33887.575,E2 33887.575} C_VEL
LIN {X 0,Y 704.299,Z 612.935,A -85,B 0,C 180,E1 33884.644,E2 33884.644} C_VEL
LIN {X 0,Y 704.32,Z 612.935,A -85,B 0,C 180,E1 33881.816,E2 33881.816} C_VEL
LIN {X 0,Y 704.256,Z 612.941,A -85,B 0,C 180,E1 33878.866,E2 33878.866} C_VEL
LIN {X 0,Y 704.288,Z 613.003,A -85,B 0,C 180,E1 33878.163,E2 33878.163} C_VEL
LIN {X 0,Y 706.261,Z 621.413,A -85,B 0,C 180,E1 33877.498,E2 33877.498} C_VEL
LIN {X 0,Y 706.087,Z 666.858,A -85,B 0,C 180,E1 33874.254,E2 33874.254} C_VEL
LIN {X 0,Y 705.853,Z 707.108,A -85,B 0,C 180,E1 33871.369,E2 33871.369} C_VEL
LIN {X 0,Y 705.574,Z 747.48,A -85,B 0,C 180,E1 33868.478,E2 33868.478} C_VEL
LIN {X 0,Y 705.205,Z 782.039,A -85,B 0,C 180,E1 33865.982,E2 33865.982} C_VEL
LIN {X 0,Y 704.848,Z 815.904,A -85,B 0,C 180,E1 33863.548,E2 33863.548} C_VEL
LIN {X 0,Y 705.319,Z 824.238,A -85,B 0,C 180,E1 33863.451,E2 33863.451} C_VEL
LIN {X 0,Y 705.03,Z 957.286,A -85,B 0,C 180,E1 33862.07,E2 33862.07} C_VEL
LIN {X 0,Y 704.92,Z 972.372,A -85,B 0,C 180,E1 33861.77,E2 33861.77} C_VEL
LIN {X 0,Y 704.807,Z 987.54,A -85,B 0,C 180,E1 33861.337,E2 33861.337} C_VEL
LIN {X 0,Y 704.617,Z 1002.557,A -85,B 0,C 180,E1 33860.737,E2 33860.737} C_VEL
LIN {X 0,Y 704.479,Z 1015.213,A -85,B 0,C 180,E1 33860.087,E2 33860.087} C_VEL
LIN {X 0,Y 704.357,Z 1025.694,A -85,B 0,C 180,E1 33859.436,E2 33859.436} C_VEL
LIN {X 0,Y 704.242,Z 1035.445,A -85,B 0,C 180,E1 33858.714,E2 33858.714} C_VEL
LIN {X 0,Y 704.147,Z 1044.219,A -85,B 0,C 180,E1 33857.943,E2 33857.943} C_VEL
LIN {X 0,Y 704.063,Z 1052.331,A -85,B 0,C 180,E1 33857.094,E2 33857.094} C_VEL
LIN {X 0,Y 703.999,Z 1059.717,A -85,B 0,C 180,E1 33856.161,E2 33856.161} C_VEL
LIN {X 0,Y 703.962,Z 1065.75,A -85,B 0,C 180,E1 33855.232,E2 33855.232} C_VEL
LIN {X 0,Y 703.935,Z 1070.981,A -85,B 0,C 180,E1 33854.223,E2 33854.223} C_VEL
LIN {X 0,Y 703.924,Z 1074.968,A -85,B 0,C 180,E1 33853.218,E2 33853.218} C_VEL
LIN {X 0,Y 703.918,Z 1077.82,A -85,B 0,C 180,E1 33852.217,E2 33852.217} C_VEL
LIN {X 0,Y 703.916,Z 1079.703,A -85,B 0,C 180,E1 33851.137,E2 33851.137} C_VEL
LIN {X 0,Y 703.917,Z 1080.399,A -85,B 0,C 180,E1 33850.06,E2 33850.06} C_VEL
LIN {X 0,Y 703.917,Z 1079.932,A -85,B 0,C 180,E1 33848.987,E2 33848.987} C_VEL
LIN {X 0,Y 703.917,Z 1078.305,A -85,B 0,C 180,E1 33847.918,E2 33847.918} C_VEL
LIN {X 0,Y 703.92,Z 1075.48,A -85,B 0,C 180,E1 33846.849,E2 33846.849} C_VEL
LIN {X 0,Y 703.929,Z 1071.784,A -85,B 0,C 180,E1 33845.868,E2 33845.868} C_VEL
LIN {X 0,Y 703.952,Z 1066.937,A -85,B 0,C 180,E1 33844.887,E2 33844.887} C_VEL
LIN {X 0,Y 703.987,Z 1061.401,A -85,B 0,C 180,E1 33843.989,E2 33843.989} C_VEL
LIN {X 0,Y 704.037,Z 1054.671,A -85,B 0,C 180,E1 33843.092,E2 33843.092} C_VEL
LIN {X 0,Y 704.118,Z 1046.538,A -85,B 0,C 180,E1 33842.196,E2 33842.196} C_VEL
LIN {X 0,Y 704.207,Z 1038.657,A -85,B 0,C 180,E1 33841.463,E2 33841.463} C_VEL
LIN {X 0,Y 704.319,Z 1028.79,A -85,B 0,C 180,E1 33840.69,E2 33840.69} C_VEL
LIN {X 0,Y 704.441,Z 1018.213,A -85,B 0,C 180,E1 33839.998,E2 33839.998} C_VEL
LIN {X 0,Y 704.53,Z 1007.868,A -85,B 0,C 180,E1 33839.429,E2 33839.429} C_VEL
LIN {X 0,Y 704.675,Z 996.166,A -85,B 0,C 180,E1 33838.901,E2 33838.901} C_VEL
LIN {X 0,Y 704.822,Z 984.966,A -85,B 0,C 180,E1 33838.494,E2 33838.494} C_VEL
LIN {X 0,Y 704.93,Z 972.176,A -85,B 0,C 180,E1 33838.136,E2 33838.136} C_VEL
LIN {X 0,Y 705.029,Z 957.568,A -85,B 0,C 180,E1 33837.844,E2 33837.844} C_VEL
LIN {X 0,Y 705.21,Z 861.519,A -85,B 0,C 180,E1 33836.841,E2 33836.841} C_VEL
LIN {X 0,Y 705.09,Z 817.797,A -85,B 0,C 180,E1 33836.387,E2 33836.387} C_VEL
LIN {X 0,Y 704.894,Z 815.689,A -85,B 0,C 180,E1 33836.339,E2 33836.339} C_VEL
LIN {X 0,Y 705.356,Z 775.226,A -85,B 0,C 180,E1 33833.405,E2 33833.405} C_VEL
LIN {X 0,Y 705.575,Z 739.025,A -85,B 0,C 180,E1 33830.825,E2 33830.825} C_VEL
LIN {X 0,Y 705.748,Z 703.823,A -85,B 0,C 180,E1 33828.351,E2 33828.351} C_VEL
LIN {X 0,Y 705.71,Z 666.95,A -85,B 0,C 180,E1 33825.81,E2 33825.81} C_VEL
LIN {X 0,Y 705.524,Z 622.066,A -85,B 0,C 180,E1 33822.811,E2 33822.811} C_VEL
LIN {X 0,Y 705.245,Z 616.915,A -85,B 0,C 180,E1 33822.464,E2 33822.464} C_VEL
LIN {X 0,Y 704.34,Z 612.935,A -85,B 0,C 180,E1 33822.185,E2 33822.185} C_VEL
LIN {X 0,Y 704.297,Z 612.938,A -85,B 0,C 180,E1 33819.088,E2 33819.088} C_VEL
LIN {X 0,Y 704.301,Z 612.939,A -85,B 0,C 180,E1 33816.398,E2 33816.398} C_VEL
LIN {X 0,Y 704.334,Z 612.935,A -85,B 0,C 180,E1 33813.345,E2 33813.345} C_VEL
LIN {X 0,Y 704.324,Z 612.938,A -85,B 0,C 180,E1 33810.392,E2 33810.392} C_VEL
LIN {X 0,Y 704.342,Z 612.937,A -85,B 0,C 180,E1 33807.449,E2 33807.449} C_VEL
LIN {X 0,Y 704.328,Z 612.937,A -85,B 0,C 180,E1 33804.504,E2 33804.504} C_VEL
LIN {X 0,Y 704.344,Z 612.932,A -85,B 0,C 180,E1 33801.448,E2 33801.448} C_VEL
LIN {X 0,Y 704.295,Z 612.937,A -85,B 0,C 180,E1 33798.43,E2 33798.43} C_VEL
LIN {X 0,Y 704.321,Z 612.935,A -85,B 0,C 180,E1 33795.566,E2 33795.566} C_VEL
LIN {X 0,Y 704.327,Z 612.935,A -85,B 0,C 180,E1 33792.51,E2 33792.51} C_VEL
LIN {X 0,Y 704.331,Z 612.938,A -85,B 0,C 180,E1 33789.568,E2 33789.568} C_VEL
LIN {X 0,Y 704.334,Z 612.938,A -85,B 0,C 180,E1 33786.599,E2 33786.599} C_VEL
LIN {X 0,Y 704.331,Z 612.938,A -85,B 0,C 180,E1 33783.704,E2 33783.704} C_VEL
LIN {X 0,Y 704.356,Z 613.042,A -85,B 0,C 180,E1 33782.947,E2 33782.947} C_VEL
LIN {X 0,Y 708.384,Z 626.81,A -85,B 0,C 180,E1 33781.663,E2 33781.663} C_VEL
LIN {X 0,Y 707.727,Z 662.203,A -85,B 0,C 180,E1 33778.938,E2 33778.938} C_VEL
LIN {X 0,Y 707.405,Z 683.292,A -85,B 0,C 180,E1 33777.358,E2 33777.358} C_VEL
LIN {X 0,Y 709.526,Z 694.112,A -85,B 0,C 180,E1 33777.149,E2 33777.149} C_VEL
LIN {X 0,Y 708.357,Z 976.73,A -85,B 0,C 180,E1 33774.079,E2 33774.079} C_VEL
LIN {X 0,Y 708.167,Z 998.018,A -85,B 0,C 180,E1 33773.768,E2 33773.768} C_VEL
LIN {X 0,Y 707.845,Z 1019.873,A -85,B 0,C 180,E1 33773.3,E2 33773.3} C_VEL
LIN {X 0,Y 707.497,Z 1041.206,A -85,B 0,C 180,E1 33772.693,E2 33772.693} C_VEL
LIN {X 0,Y 707.088,Z 1061.669,A -85,B 0,C 180,E1 33771.958,E2 33771.958} C_VEL
LIN {X 0,Y 706.648,Z 1081.093,A -85,B 0,C 180,E1 33771.105,E2 33771.105} C_VEL
LIN {X 0,Y 706.19,Z 1100.741,A -85,B 0,C 180,E1 33770.08,E2 33770.08} C_VEL
LIN {X 0,Y 705.737,Z 1119.415,A -85,B 0,C 180,E1 33768.931,E2 33768.931} C_VEL
LIN {X 0,Y 705.309,Z 1136.911,A -85,B 0,C 180,E1 33767.659,E2 33767.659} C_VEL
LIN {X 0,Y 704.943,Z 1152.878,A -85,B 0,C 180,E1 33766.309,E2 33766.309} C_VEL
LIN {X 0,Y 704.649,Z 1167.471,A -85,B 0,C 180,E1 33764.881,E2 33764.881} C_VEL
LIN {X 0,Y 704.394,Z 1180.676,A -85,B 0,C 180,E1 33763.377,E2 33763.377} C_VEL
LIN {X 0,Y 704.198,Z 1192.399,A -85,B 0,C 180,E1 33761.797,E2 33761.797} C_VEL
LIN {X 0,Y 704.067,Z 1203.221,A -85,B 0,C 180,E1 33760.059,E2 33760.059} C_VEL
LIN {X 0,Y 704.001,Z 1211.703,A -85,B 0,C 180,E1 33758.411,E2 33758.411} C_VEL
LIN {X 0,Y 703.931,Z 1218.676,A -85,B 0,C 180,E1 33756.688,E2 33756.688} C_VEL
LIN {X 0,Y 703.905,Z 1224.2,A -85,B 0,C 180,E1 33754.888,E2 33754.888} C_VEL
LIN {X 0,Y 703.9,Z 1227.881,A -85,B 0,C 180,E1 33753.175,E2 33753.175} C_VEL
LIN {X 0,Y 703.899,Z 1229.884,A -85,B 0,C 180,E1 33751.464,E2 33751.464} C_VEL
LIN {X 0,Y 703.898,Z 1230.396,A -85,B 0,C 180,E1 33749.592,E2 33749.592} C_VEL
LIN {X 0,Y 703.914,Z 1229.23,A -85,B 0,C 180,E1 33747.801,E2 33747.801} C_VEL
LIN {X 0,Y 703.918,Z 1226.303,A -85,B 0,C 180,E1 33746.008,E2 33746.008} C_VEL
LIN {X 0,Y 703.918,Z 1221.65,A -85,B 0,C 180,E1 33744.211,E2 33744.211} C_VEL
LIN {X 0,Y 703.953,Z 1215.58,A -85,B 0,C 180,E1 33742.49,E2 33742.49} C_VEL
LIN {X 0,Y 704.017,Z 1208.062,A -85,B 0,C 180,E1 33740.846,E2 33740.846} C_VEL
LIN {X 0,Y 704.119,Z 1198.321,A -85,B 0,C 180,E1 33739.112,E2 33739.112} C_VEL
LIN {X 0,Y 704.286,Z 1187.718,A -85,B 0,C 180,E1 33737.537,E2 33737.537} C_VEL
LIN {X 0,Y 704.496,Z 1175.035,A -85,B 0,C 180,E1 33735.953,E2 33735.953} C_VEL
LIN {X 0,Y 704.754,Z 1161.703,A -85,B 0,C 180,E1 33734.529,E2 33734.529} C_VEL
LIN {X 0,Y 705.09,Z 1146.187,A -85,B 0,C 180,E1 33733.099,E2 33733.099} C_VEL
LIN {X 0,Y 705.49,Z 1129.676,A -85,B 0,C 180,E1 33731.788,E2 33731.788} C_VEL
LIN {X 0,Y 705.905,Z 1112.512,A -85,B 0,C 180,E1 33730.626,E2 33730.626} C_VEL
LIN {X 0,Y 706.371,Z 1092.922,A -85,B 0,C 180,E1 33729.491,E2 33729.491} C_VEL
LIN {X 0,Y 706.829,Z 1073.392,A -85,B 0,C 180,E1 33728.536,E2 33728.536} C_VEL
LIN {X 0,Y 707.26,Z 1053.613,A -85,B 0,C 180,E1 33727.735,E2 33727.735} C_VEL
LIN {X 0,Y 707.622,Z 1032.65,A -85,B 0,C 180,E1 33727.045,E2 33727.045} C_VEL
LIN {X 0,Y 708.004,Z 1010.92,A -85,B 0,C 180,E1 33726.489,E2 33726.489} C_VEL
LIN {X 0,Y 708.243,Z 989.77,A -85,B 0,C 180,E1 33726.094,E2 33726.094} C_VEL
LIN {X 0,Y 708.464,Z 956.42,A -85,B 0,C 180,E1 33725.699,E2 33725.699} C_VEL
LIN {X 0,Y 709.482,Z 692.744,A -85,B 0,C 180,E1 33722.834,E2 33722.834} C_VEL
LIN {X 0,Y 707.334,Z 682.778,A -85,B 0,C 180,E1 33722.627,E2 33722.627} C_VEL
LIN {X 0,Y 708.095,Z 644.233,A -85,B 0,C 180,E1 33719.68,E2 33719.68} C_VEL
LIN {X 0,Y 708.12,Z 625.43,A -85,B 0,C 180,E1 33718.265,E2 33718.265} C_VEL
LIN {X 0,Y 704.339,Z 612.933,A -85,B 0,C 180,E1 33717.135,E2 33717.135} C_VEL
LIN {X 0,Y 704.326,Z 612.938,A -85,B 0,C 180,E1 33714.003,E2 33714.003} C_VEL
LIN {X 0,Y 704.333,Z 612.929,A -85,B 0,C 180,E1 33711.031,E2 33711.031} C_VEL
LIN {X 0,Y 704.324,Z 612.938,A -85,B 0,C 180,E1 33707.927,E2 33707.927} C_VEL
LIN {X 0,Y 704.317,Z 612.93,A -85,B 0,C 180,E1 33704.992,E2 33704.992} C_VEL
LIN {X 0,Y 704.32,Z 612.938,A -85,B 0,C 180,E1 33701.855,E2 33701.855} C_VEL
LIN {X 0,Y 704.295,Z 612.933,A -85,B 0,C 180,E1 33699.051,E2 33699.051} C_VEL
LIN {X 0,Y 704.344,Z 612.936,A -85,B 0,C 180,E1 33696.097,E2 33696.097} C_VEL
LIN {X 0,Y 704.28,Z 612.937,A -85,B 0,C 180,E1 33693.232,E2 33693.232} C_VEL
LIN {X 0,Y 704.329,Z 612.934,A -85,B 0,C 180,E1 33690.453,E2 33690.453} C_VEL
LIN {X 0,Y 704.318,Z 612.956,A -85,B 0,C 180,E1 33688.468,E2 33688.468} C_VEL
LIN {X 0,Y 706.819,Z 623.895,A -85,B 0,C 180,E1 33687.349,E2 33687.349} C_VEL
LIN {X 0,Y 709.519,Z 635.778,A -85,B 0,C 180,E1 33687.085,E2 33687.085} C_VEL
LIN {X 0,Y 708.455,Z 898.815,A -85,B 0,C 180,E1 33684.23,E2 33684.23} C_VEL
LIN {X 0,Y 708.244,Z 930.275,A -85,B 0,C 180,E1 33683.853,E2 33683.853} C_VEL
LIN {X 0,Y 708.005,Z 952.055,A -85,B 0,C 180,E1 33683.443,E2 33683.443} C_VEL
LIN {X 0,Y 707.613,Z 973.649,A -85,B 0,C 180,E1 33682.882,E2 33682.882} C_VEL
LIN {X 0,Y 707.219,Z 994.945,A -85,B 0,C 180,E1 33682.171,E2 33682.171} C_VEL
LIN {X 0,Y 706.811,Z 1014.651,A -85,B 0,C 180,E1 33681.364,E2 33681.364} C_VEL
LIN {X 0,Y 706.33,Z 1034.517,A -85,B 0,C 180,E1 33680.381,E2 33680.381} C_VEL
LIN {X 0,Y 705.872,Z 1053.927,A -85,B 0,C 180,E1 33679.241,E2 33679.241} C_VEL
LIN {X 0,Y 705.432,Z 1071.949,A -85,B 0,C 180,E1 33677.994,E2 33677.994} C_VEL
LIN {X 0,Y 705.042,Z 1088.617,A -85,B 0,C 180,E1 33676.649,E2 33676.649} C_VEL
LIN {X 0,Y 704.717,Z 1103.812,A -85,B 0,C 180,E1 33675.219,E2 33675.219} C_VEL
LIN {X 0,Y 704.453,Z 1117.482,A -85,B 0,C 180,E1 33673.713,E2 33673.713} C_VEL
LIN {X 0,Y 704.246,Z 1130.34,A -85,B 0,C 180,E1 33672.048,E2 33672.048} C_VEL
LIN {X 0,Y 704.096,Z 1141.09,A -85,B 0,C 180,E1 33670.392,E2 33670.392} C_VEL
LIN {X 0,Y 704,Z 1149.878,A -85,B 0,C 180,E1 33668.743,E2 33668.743} C_VEL
LIN {X 0,Y 703.941,Z 1157.602,A -85,B 0,C 180,E1 33666.936,E2 33666.936} C_VEL
LIN {X 0,Y 703.931,Z 1163.243,A -85,B 0,C 180,E1 33665.217,E2 33665.217} C_VEL
LIN {X 0,Y 703.918,Z 1167.17,A -85,B 0,C 180,E1 33663.503,E2 33663.503} C_VEL
LIN {X 0,Y 703.914,Z 1169.713,A -85,B 0,C 180,E1 33661.63,E2 33661.63} C_VEL
LIN {X 0,Y 703.91,Z 1170.475,A -85,B 0,C 180,E1 33659.839,E2 33659.839} C_VEL
LIN {X 0,Y 703.912,Z 1169.586,A -85,B 0,C 180,E1 33658.13,E2 33658.13} C_VEL
LIN {X 0,Y 703.915,Z 1167.037,A -85,B 0,C 180,E1 33656.337,E2 33656.337} C_VEL
LIN {X 0,Y 703.929,Z 1162.82,A -85,B 0,C 180,E1 33654.541,E2 33654.541} C_VEL
LIN {X 0,Y 703.956,Z 1157.032,A -85,B 0,C 180,E1 33652.822,E2 33652.822} C_VEL
LIN {X 0,Y 704.016,Z 1149.123,A -85,B 0,C 180,E1 33651.014,E2 33651.014} C_VEL
LIN {X 0,Y 704.112,Z 1139.937,A -85,B 0,C 180,E1 33649.324,E2 33649.324} C_VEL
LIN {X 0,Y 704.26,Z 1129.243,A -85,B 0,C 180,E1 33647.706,E2 33647.706} C_VEL
LIN {X 0,Y 704.467,Z 1116.861,A -85,B 0,C 180,E1 33646.123,E2 33646.123} C_VEL
LIN {X 0,Y 704.733,Z 1103.059,A -85,B 0,C 180,E1 33644.616,E2 33644.616} C_VEL
LIN {X 0,Y 705.071,Z 1087.288,A -85,B 0,C 180,E1 33643.144,E2 33643.144} C_VEL
LIN {X 0,Y 705.47,Z 1070.277,A -85,B 0,C 180,E1 33641.791,E2 33641.791} C_VEL
LIN {X 0,Y 705.853,Z 1054.615,A -85,B 0,C 180,E1 33640.713,E2 33640.713} C_VEL
LIN {X 0,Y 705.065,Z 1048.697,A -85,B 0,C 180,E1 33640.313,E2 33640.313} C_VEL
LIN {X 0,Y 699.546,Z 1032.974,A -85,B 0,C 180,E1 33639.237,E2 33639.237} C_VEL
LIN {X 0,Y 698.921,Z 1027.536,A -85,B 0,C 180,E1 33638.928,E2 33638.928} C_VEL
LIN {X 0,Y 699.433,Z 1007.819,A -85,B 0,C 180,E1 33638.006,E2 33638.006} C_VEL
LIN {X 0,Y 699.916,Z 987.709,A -85,B 0,C 180,E1 33637.225,E2 33637.225} C_VEL
LIN {X 0,Y 700.386,Z 966.328,A -85,B 0,C 180,E1 33636.56,E2 33636.56} C_VEL
LIN {X 0,Y 700.712,Z 944.697,A -85,B 0,C 180,E1 33636.051,E2 33636.051} C_VEL
LIN {X 0,Y 701.01,Z 921.94,A -85,B 0,C 180,E1 33635.675,E2 33635.675} C_VEL
LIN {X 0,Y 702.395,Z 645.496,A -85,B 0,C 180,E1 33632.636,E2 33632.636} C_VEL
LIN {X 0,Y 702.219,Z 635.693,A -85,B 0,C 180,E1 33632.518,E2 33632.518} C_VEL
LIN {X 0,Y 699.025,Z 624.07,A -85,B 0,C 180,E1 33632.245,E2 33632.245} C_VEL
LIN {X 0,Y 696.357,Z 613.926,A -85,B 0,C 180,E1 33631.151,E2 33631.151} C_VEL
LIN {X 0,Y 696.341,Z 613.93,A -85,B 0,C 180,E1 33628.063,E2 33628.063} C_VEL
LIN {X 0,Y 696.332,Z 613.928,A -85,B 0,C 180,E1 33625.366,E2 33625.366} C_VEL
LIN {X 0,Y 696.397,Z 613.918,A -85,B 0,C 180,E1 33622.398,E2 33622.398} C_VEL
LIN {X 0,Y 696.389,Z 613.924,A -85,B 0,C 180,E1 33619.425,E2 33619.425} C_VEL
LIN {X 0,Y 696.401,Z 613.916,A -85,B 0,C 180,E1 33616.325,E2 33616.325} C_VEL
LIN {X 0,Y 696.355,Z 613.925,A -85,B 0,C 180,E1 33613.285,E2 33613.285} C_VEL
LIN {X 0,Y 696.333,Z 613.926,A -85,B 0,C 180,E1 33610.687,E2 33610.687} C_VEL
LIN {X 0,Y 696.336,Z 613.925,A -85,B 0,C 180,E1 33607.506,E2 33607.506} C_VEL
LIN {X 0,Y 696.361,Z 613.924,A -85,B 0,C 180,E1 33604.854,E2 33604.854} C_VEL
LIN {X 0,Y 696.399,Z 613.916,A -85,B 0,C 180,E1 33601.794,E2 33601.794} C_VEL
LIN {X 0,Y 696.389,Z 613.925,A -85,B 0,C 180,E1 33598.751,E2 33598.751} C_VEL
LIN {X 0,Y 696.395,Z 613.918,A -85,B 0,C 180,E1 33595.789,E2 33595.789} C_VEL
LIN {X 0,Y 696.326,Z 613.925,A -85,B 0,C 180,E1 33592.805,E2 33592.805} C_VEL
LIN {X 0,Y 696.33,Z 613.927,A -85,B 0,C 180,E1 33590.247,E2 33590.247} C_VEL
LIN {X 0,Y 696.364,Z 613.92,A -85,B 0,C 180,E1 33587.12,E2 33587.12} C_VEL
LIN {X 0,Y 696.402,Z 613.924,A -85,B 0,C 180,E1 33584.214,E2 33584.214} C_VEL
LIN {X 0,Y 696.4,Z 613.917,A -85,B 0,C 180,E1 33581.177,E2 33581.177} C_VEL
LIN {X 0,Y 696.363,Z 613.922,A -85,B 0,C 180,E1 33578.256,E2 33578.256} C_VEL
LIN {X 0,Y 696.353,Z 613.924,A -85,B 0,C 180,E1 33575.522,E2 33575.522} C_VEL
LIN {X 0,Y 696.325,Z 613.923,A -85,B 0,C 180,E1 33572.47,E2 33572.47} C_VEL
LIN {X 0,Y 696.353,Z 613.925,A -85,B 0,C 180,E1 33569.837,E2 33569.837} C_VEL
LIN {X 0,Y 696.394,Z 613.914,A -85,B 0,C 180,E1 33566.791,E2 33566.791} C_VEL
LIN {X 0,Y 696.393,Z 613.924,A -85,B 0,C 180,E1 33563.737,E2 33563.737} C_VEL
LIN {X 0,Y 696.401,Z 613.917,A -85,B 0,C 180,E1 33560.747,E2 33560.747} C_VEL
LIN {X 0,Y 696.338,Z 613.923,A -85,B 0,C 180,E1 33557.816,E2 33557.816} C_VEL
LIN {X 0,Y 696.321,Z 613.927,A -85,B 0,C 180,E1 33555.277,E2 33555.277} C_VEL
LIN {X 0,Y 696.364,Z 613.921,A -85,B 0,C 180,E1 33552.193,E2 33552.193} C_VEL
LIN {X 0,Y 696.384,Z 613.924,A -85,B 0,C 180,E1 33549.318,E2 33549.318} C_VEL
LIN {X 0,Y 696.398,Z 613.916,A -85,B 0,C 180,E1 33546.207,E2 33546.207} C_VEL
LIN {X 0,Y 696.369,Z 613.924,A -85,B 0,C 180,E1 33543.203,E2 33543.203} C_VEL
LIN {X 0,Y 696.373,Z 613.922,A -85,B 0,C 180,E1 33540.402,E2 33540.402} C_VEL
LIN {X 0,Y 696.323,Z 613.927,A -85,B 0,C 180,E1 33537.421,E2 33537.421} C_VEL
LIN {X 0,Y 696.342,Z 613.926,A -85,B 0,C 180,E1 33534.846,E2 33534.846} C_VEL
LIN {X 0,Y 696.388,Z 613.918,A -85,B 0,C 180,E1 33531.771,E2 33531.771} C_VEL
LIN {X 0,Y 696.403,Z 613.925,A -85,B 0,C 180,E1 33528.777,E2 33528.777} C_VEL
LIN {X 0,Y 696.404,Z 613.917,A -85,B 0,C 180,E1 33525.752,E2 33525.752} C_VEL
LIN {X 0,Y 696.346,Z 613.927,A -85,B 0,C 180,E1 33522.776,E2 33522.776} C_VEL
LIN {X 0,Y 696.325,Z 613.929,A -85,B 0,C 180,E1 33520.191,E2 33520.191} C_VEL
LIN {X 0,Y 696.341,Z 614.058,A -85,B 0,C 180,E1 33518.362,E2 33518.362} C_VEL
LIN {X 0,Y 698.619,Z 623.346,A -85,B 0,C 180,E1 33517.617,E2 33517.617} C_VEL
LIN {X 0,Y 698.421,Z 666.95,A -85,B 0,C 180,E1 33514.494,E2 33514.494} C_VEL
LIN {X 0,Y 698.157,Z 706.998,A -85,B 0,C 180,E1 33511.61,E2 33511.61} C_VEL
LIN {X 0,Y 697.833,Z 746.898,A -85,B 0,C 180,E1 33508.733,E2 33508.733} C_VEL
LIN {X 0,Y 697.433,Z 783.557,A -85,B 0,C 180,E1 33506.08,E2 33506.08} C_VEL
LIN {X 0,Y 697.094,Z 816.81,A -85,B 0,C 180,E1 33503.693,E2 33503.693} C_VEL
LIN {X 0,Y 697.539,Z 825.005,A -85,B 0,C 180,E1 33503.597,E2 33503.597} C_VEL
LIN {X 0,Y 697.195,Z 958.266,A -85,B 0,C 180,E1 33502.19,E2 33502.19} C_VEL
LIN {X 0,Y 697.085,Z 974.09,A -85,B 0,C 180,E1 33501.87,E2 33501.87} C_VEL
LIN {X 0,Y 696.94,Z 990.698,A -85,B 0,C 180,E1 33501.369,E2 33501.369} C_VEL
LIN {X 0,Y 696.761,Z 1004.099,A -85,B 0,C 180,E1 33500.813,E2 33500.813} C_VEL
LIN {X 0,Y 696.617,Z 1016.406,A -85,B 0,C 180,E1 33500.168,E2 33500.168} C_VEL
LIN {X 0,Y 696.47,Z 1026.94,A -85,B 0,C 180,E1 33499.497,E2 33499.497} C_VEL
LIN {X 0,Y 696.329,Z 1036.586,A -85,B 0,C 180,E1 33498.761,E2 33498.761} C_VEL
LIN {X 0,Y 696.212,Z 1045.146,A -85,B 0,C 180,E1 33497.983,E2 33497.983} C_VEL
LIN {X 0,Y 696.105,Z 1053.091,A -85,B 0,C 180,E1 33497.123,E2 33497.123} C_VEL
LIN {X 0,Y 696.03,Z 1059.708,A -85,B 0,C 180,E1 33496.266,E2 33496.266} C_VEL
LIN {X 0,Y 695.975,Z 1065.681,A -85,B 0,C 180,E1 33495.326,E2 33495.326} C_VEL
LIN {X 0,Y 695.939,Z 1070.849,A -85,B 0,C 180,E1 33494.305,E2 33494.305} C_VEL
LIN {X 0,Y 695.926,Z 1074.848,A -85,B 0,C 180,E1 33493.288,E2 33493.288} C_VEL
LIN {X 0,Y 695.919,Z 1077.737,A -85,B 0,C 180,E1 33492.275,E2 33492.275} C_VEL
LIN {X 0,Y 695.916,Z 1079.655,A -85,B 0,C 180,E1 33491.182,E2 33491.182} C_VEL
LIN {X 0,Y 695.916,Z 1080.385,A -85,B 0,C 180,E1 33490.093,E2 33490.093} C_VEL
LIN {X 0,Y 695.917,Z 1079.952,A -85,B 0,C 180,E1 33489.008,E2 33489.008} C_VEL
LIN {X 0,Y 695.918,Z 1078.359,A -85,B 0,C 180,E1 33487.926,E2 33487.926} C_VEL
LIN {X 0,Y 695.922,Z 1075.71,A -85,B 0,C 180,E1 33486.888,E2 33486.888} C_VEL
LIN {X 0,Y 695.932,Z 1071.926,A -85,B 0,C 180,E1 33485.853,E2 33485.853} C_VEL
LIN {X 0,Y 695.962,Z 1067.224,A -85,B 0,C 180,E1 33484.861,E2 33484.861} C_VEL
LIN {X 0,Y 696.015,Z 1061.28,A -85,B 0,C 180,E1 33483.87,E2 33483.87} C_VEL
LIN {X 0,Y 696.088,Z 1054.593,A -85,B 0,C 180,E1 33482.962,E2 33482.962} C_VEL
LIN {X 0,Y 696.186,Z 1047.309,A -85,B 0,C 180,E1 33482.138,E2 33482.138} C_VEL
LIN {X 0,Y 696.311,Z 1038.623,A -85,B 0,C 180,E1 33481.315,E2 33481.315} C_VEL
LIN {X 0,Y 696.456,Z 1028.733,A -85,B 0,C 180,E1 33480.533,E2 33480.533} C_VEL
LIN {X 0,Y 696.598,Z 1018.086,A -85,B 0,C 180,E1 33479.834,E2 33479.834} C_VEL
LIN {X 0,Y 696.715,Z 1006.693,A -85,B 0,C 180,E1 33479.217,E2 33479.217} C_VEL
LIN {X 0,Y 696.897,Z 993.431,A -85,B 0,C 180,E1 33478.642,E2 33478.642} C_VEL
LIN {X 0,Y 697.086,Z 976.17,A -85,B 0,C 180,E1 33478.092,E2 33478.092} C_VEL
LIN {X 0,Y 697.191,Z 959.879,A -85,B 0,C 180,E1 33477.746,E2 33477.746} C_VEL
LIN {X 0,Y 697.276,Z 921.867,A -85,B 0,C 180,E1 33477.323,E2 33477.323} C_VEL
LIN {X 0,Y 697.333,Z 818.64,A -85,B 0,C 180,E1 33476.242,E2 33476.242} C_VEL
LIN {X 0,Y 697.164,Z 817.1,A -85,B 0,C 180,E1 33476.216,E2 33476.216} C_VEL
LIN {X 0,Y 697.628,Z 773.781,A -85,B 0,C 180,E1 33473.083,E2 33473.083} C_VEL
LIN {X 0,Y 697.861,Z 737.186,A -85,B 0,C 180,E1 33470.473,E2 33470.473} C_VEL
LIN {X 0,Y 698.087,Z 699.213,A -85,B 0,C 180,E1 33467.802,E2 33467.802} C_VEL
LIN {X 0,Y 697.919,Z 659.126,A -85,B 0,C 180,E1 33465.054,E2 33465.054} C_VEL
LIN {X 0,Y 697.75,Z 619.782,A -85,B 0,C 180,E1 33462.442,E2 33462.442} C_VEL
LIN {X 0,Y 696.404,Z 613.923,A -85,B 0,C 180,E1 33461.996,E2 33461.996} C_VEL
LIN {X 0,Y 696.364,Z 613.927,A -85,B 0,C 180,E1 33458.952,E2 33458.952} C_VEL
LIN {X 0,Y 696.377,Z 613.928,A -85,B 0,C 180,E1 33456.113,E2 33456.113} C_VEL
LIN {X 0,Y 696.4,Z 613.926,A -85,B 0,C 180,E1 33453.109,E2 33453.109} C_VEL
LIN {X 0,Y 696.405,Z 613.925,A -85,B 0,C 180,E1 33450.116,E2 33450.116} C_VEL
LIN {X 0,Y 696.37,Z 613.926,A -85,B 0,C 180,E1 33447.127,E2 33447.127} C_VEL
LIN {X 0,Y 696.378,Z 613.925,A -85,B 0,C 180,E1 33444.34,E2 33444.34} C_VEL
LIN {X 0,Y 696.395,Z 613.922,A -85,B 0,C 180,E1 33441.225,E2 33441.225} C_VEL
LIN {X 0,Y 696.359,Z 613.926,A -85,B 0,C 180,E1 33438.299,E2 33438.299} C_VEL
LIN {X 0,Y 696.402,Z 613.923,A -85,B 0,C 180,E1 33435.287,E2 33435.287} C_VEL
LIN {X 0,Y 696.399,Z 613.924,A -85,B 0,C 180,E1 33432.216,E2 33432.216} C_VEL
LIN {X 0,Y 696.408,Z 613.922,A -85,B 0,C 180,E1 33429.164,E2 33429.164} C_VEL
LIN {X 0,Y 696.361,Z 613.928,A -85,B 0,C 180,E1 33426.165,E2 33426.165} C_VEL
LIN {X 0,Y 696.395,Z 613.989,A -85,B 0,C 180,E1 33423.273,E2 33423.273} C_VEL
LIN {X 0,Y 701.01,Z 628.866,A -85,B 0,C 180,E1 33421.852,E2 33421.852} C_VEL
LIN {X 0,Y 700.276,Z 665.19,A -85,B 0,C 180,E1 33419.041,E2 33419.041} C_VEL
LIN {X 0,Y 699.978,Z 683.286,A -85,B 0,C 180,E1 33417.673,E2 33417.673} C_VEL
LIN {X 0,Y 702.4,Z 695.47,A -85,B 0,C 180,E1 33417.432,E2 33417.432} C_VEL
LIN {X 0,Y 701.042,Z 977.459,A -85,B 0,C 180,E1 33414.337,E2 33414.337} C_VEL
LIN {X 0,Y 700.824,Z 998.991,A -85,B 0,C 180,E1 33414.016,E2 33414.016} C_VEL
LIN {X 0,Y 700.452,Z 1020.638,A -85,B 0,C 180,E1 33413.541,E2 33413.541} C_VEL
LIN {X 0,Y 700.03,Z 1042.489,A -85,B 0,C 180,E1 33412.905,E2 33412.905} C_VEL
LIN {X 0,Y 699.57,Z 1063.072,A -85,B 0,C 180,E1 33412.151,E2 33412.151} C_VEL
LIN {X 0,Y 699.031,Z 1083.186,A -85,B 0,C 180,E1 33411.244,E2 33411.244} C_VEL
LIN {X 0,Y 698.495,Z 1102.941,A -85,B 0,C 180,E1 33410.18,E2 33410.18} C_VEL
LIN {X 0,Y 697.974,Z 1121.466,A -85,B 0,C 180,E1 33409.003,E2 33409.003} C_VEL
LIN {X 0,Y 697.501,Z 1138.628,A -85,B 0,C 180,E1 33407.729,E2 33407.729} C_VEL
LIN {X 0,Y 697.096,Z 1153.804,A -85,B 0,C 180,E1 33406.412,E2 33406.412} C_VEL
LIN {X 0,Y 696.735,Z 1169.022,A -85,B 0,C 180,E1 33404.884,E2 33404.884} C_VEL
LIN {X 0,Y 696.453,Z 1182,A -85,B 0,C 180,E1 33403.363,E2 33403.363} C_VEL
LIN {X 0,Y 696.234,Z 1193.544,A -85,B 0,C 180,E1 33401.766,E2 33401.766} C_VEL
LIN {X 0,Y 696.089,Z 1203.682,A -85,B 0,C 180,E1 33400.092,E2 33400.092} C_VEL
LIN {X 0,Y 696.008,Z 1212.41,A -85,B 0,C 180,E1 33398.342,E2 33398.342} C_VEL
LIN {X 0,Y 695.935,Z 1218.978,A -85,B 0,C 180,E1 33396.682,E2 33396.682} C_VEL
LIN {X 0,Y 695.908,Z 1224.2,A -85,B 0,C 180,E1 33394.944,E2 33394.944} C_VEL
LIN {X 0,Y 695.901,Z 1227.881,A -85,B 0,C 180,E1 33393.211,E2 33393.211} C_VEL
LIN {X 0,Y 695.9,Z 1229.884,A -85,B 0,C 180,E1 33391.481,E2 33391.481} C_VEL
LIN {X 0,Y 695.899,Z 1230.396,A -85,B 0,C 180,E1 33389.587,E2 33389.587} C_VEL
LIN {X 0,Y 695.914,Z 1229.231,A -85,B 0,C 180,E1 33387.776,E2 33387.776} C_VEL
LIN {X 0,Y 695.92,Z 1226.302,A -85,B 0,C 180,E1 33385.962,E2 33385.962} C_VEL
LIN {X 0,Y 695.922,Z 1221.651,A -85,B 0,C 180,E1 33384.144,E2 33384.144} C_VEL
LIN {X 0,Y 695.961,Z 1215.58,A -85,B 0,C 180,E1 33382.404,E2 33382.404} C_VEL
LIN {X 0,Y 696.035,Z 1207.977,A -85,B 0,C 180,E1 33380.723,E2 33380.723} C_VEL
LIN {X 0,Y 696.157,Z 1198.32,A -85,B 0,C 180,E1 33378.986,E2 33378.986} C_VEL
LIN {X 0,Y 696.347,Z 1187.717,A -85,B 0,C 180,E1 33377.392,E2 33377.392} C_VEL
LIN {X 0,Y 696.595,Z 1175.036,A -85,B 0,C 180,E1 33375.79,E2 33375.79} C_VEL
LIN {X 0,Y 696.91,Z 1161.268,A -85,B 0,C 180,E1 33374.307,E2 33374.307} C_VEL
LIN {X 0,Y 697.309,Z 1145.684,A -85,B 0,C 180,E1 33372.862,E2 33372.862} C_VEL
LIN {X 0,Y 697.763,Z 1129.09,A -85,B 0,C 180,E1 33371.536,E2 33371.536} C_VEL
LIN {X 0,Y 698.261,Z 1111.417,A -85,B 0,C 180,E1 33370.335,E2 33370.335} C_VEL
LIN {X 0,Y 698.769,Z 1093.043,A -85,B 0,C 180,E1 33369.264,E2 33369.264} C_VEL
LIN {X 0,Y 699.284,Z 1073.809,A -85,B 0,C 180,E1 33368.311,E2 33368.311} C_VEL
LIN {X 0,Y 699.791,Z 1053.609,A -85,B 0,C 180,E1 33367.484,E2 33367.484} C_VEL
LIN {X 0,Y 700.214,Z 1032.648,A -85,B 0,C 180,E1 33366.788,E2 33366.788} C_VEL
LIN {X 0,Y 700.643,Z 1010.922,A -85,B 0,C 180,E1 33366.226,E2 33366.226} C_VEL
LIN {X 0,Y 700.927,Z 989.607,A -85,B 0,C 180,E1 33365.826,E2 33365.826} C_VEL
LIN {X 0,Y 701.177,Z 955.366,A -85,B 0,C 180,E1 33365.419,E2 33365.419} C_VEL
LIN {X 0,Y 702.368,Z 694.229,A -85,B 0,C 180,E1 33362.553,E2 33362.553} C_VEL
LIN {X 0,Y 699.915,Z 682.539,A -85,B 0,C 180,E1 33362.293,E2 33362.293} C_VEL
LIN {X 0,Y 700.514,Z 650.266,A -85,B 0,C 180,E1 33359.838,E2 33359.838} C_VEL
LIN {X 0,Y 700.55,Z 627.785,A -85,B 0,C 180,E1 33358.13,E2 33358.13} C_VEL
LIN {X 0,Y 696.396,Z 613.925,A -85,B 0,C 180,E1 33356.86,E2 33356.86} C_VEL
LIN {X 0,Y 696.377,Z 613.927,A -85,B 0,C 180,E1 33353.833,E2 33353.833} C_VEL
LIN {X 0,Y 696.402,Z 613.918,A -85,B 0,C 180,E1 33350.836,E2 33350.836} C_VEL
LIN {X 0,Y 696.373,Z 613.926,A -85,B 0,C 180,E1 33347.779,E2 33347.779} C_VEL
LIN {X 0,Y 696.394,Z 613.918,A -85,B 0,C 180,E1 33344.822,E2 33344.822} C_VEL
LIN {X 0,Y 696.373,Z 613.927,A -85,B 0,C 180,E1 33341.778,E2 33341.778} C_VEL
LIN {X 0,Y 696.362,Z 613.922,A -85,B 0,C 180,E1 33338.971,E2 33338.971} C_VEL
LIN {X 0,Y 696.393,Z 613.927,A -85,B 0,C 180,E1 33335.923,E2 33335.923} C_VEL
LIN {X 0,Y 696.341,Z 613.926,A -85,B 0,C 180,E1 33333.16,E2 33333.16} C_VEL
LIN {X 0,Y 696.409,Z 613.924,A -85,B 0,C 180,E1 33330.264,E2 33330.264} C_VEL
LIN {X 0,Y 696.348,Z 613.945,A -85,B 0,C 180,E1 33328.754,E2 33328.754} C_VEL
LIN {X 0,Y 699.097,Z 624.487,A -85,B 0,C 180,E1 33327.652,E2 33327.652} C_VEL
LIN {X 0,Y 702.393,Z 636.465,A -85,B 0,C 180,E1 33327.376,E2 33327.376} C_VEL
LIN {X 0,Y 701.158,Z 899.503,A -85,B 0,C 180,E1 33324.491,E2 33324.491} C_VEL
LIN {X 0,Y 700.922,Z 930.386,A -85,B 0,C 180,E1 33324.116,E2 33324.116} C_VEL
LIN {X 0,Y 700.641,Z 952.218,A -85,B 0,C 180,E1 33323.702,E2 33323.702} C_VEL
LIN {X 0,Y 700.218,Z 972.793,A -85,B 0,C 180,E1 33323.164,E2 33323.164} C_VEL
LIN {X 0,Y 699.754,Z 994.708,A -85,B 0,C 180,E1 33322.429,E2 33322.429} C_VEL
LIN {X 0,Y 699.268,Z 1014.656,A -85,B 0,C 180,E1 33321.606,E2 33321.606} C_VEL
LIN {X 0,Y 698.728,Z 1034.534,A -85,B 0,C 180,E1 33320.613,E2 33320.613} C_VEL
LIN {X 0,Y 698.188,Z 1054.101,A -85,B 0,C 180,E1 33319.45,E2 33319.45} C_VEL
LIN {X 0,Y 697.667,Z 1072.539,A -85,B 0,C 180,E1 33318.157,E2 33318.157} C_VEL
LIN {X 0,Y 697.204,Z 1089.567,A -85,B 0,C 180,E1 33316.755,E2 33316.755} C_VEL
LIN {X 0,Y 696.837,Z 1104.653,A -85,B 0,C 180,E1 33315.31,E2 33315.31} C_VEL
LIN {X 0,Y 696.533,Z 1118.195,A -85,B 0,C 180,E1 33313.788,E2 33313.788} C_VEL
LIN {X 0,Y 696.294,Z 1130.926,A -85,B 0,C 180,E1 33312.104,E2 33312.104} C_VEL
LIN {X 0,Y 696.121,Z 1141.558,A -85,B 0,C 180,E1 33310.429,E2 33310.429} C_VEL
LIN {X 0,Y 696.014,Z 1150.289,A -85,B 0,C 180,E1 33308.761,E2 33308.761} C_VEL
LIN {X 0,Y 695.952,Z 1157.606,A -85,B 0,C 180,E1 33307.016,E2 33307.016} C_VEL
LIN {X 0,Y 695.93,Z 1163.453,A -85,B 0,C 180,E1 33305.195,E2 33305.195} C_VEL
LIN {X 0,Y 695.918,Z 1167.329,A -85,B 0,C 180,E1 33303.461,E2 33303.461} C_VEL
LIN {X 0,Y 695.914,Z 1169.713,A -85,B 0,C 180,E1 33301.648,E2 33301.648} C_VEL
LIN {X 0,Y 695.91,Z 1170.474,A -85,B 0,C 180,E1 33299.837,E2 33299.837} C_VEL
LIN {X 0,Y 695.911,Z 1169.585,A -85,B 0,C 180,E1 33298.108,E2 33298.108} C_VEL
LIN {X 0,Y 695.914,Z 1167.038,A -85,B 0,C 180,E1 33296.295,E2 33296.295} C_VEL
LIN {X 0,Y 695.928,Z 1162.821,A -85,B 0,C 180,E1 33294.478,E2 33294.478} C_VEL
LIN {X 0,Y 695.966,Z 1157.029,A -85,B 0,C 180,E1 33292.739,E2 33292.739} C_VEL
LIN {X 0,Y 696.035,Z 1149.123,A -85,B 0,C 180,E1 33290.91,E2 33290.91} C_VEL
LIN {X 0,Y 696.144,Z 1140.181,A -85,B 0,C 180,E1 33289.24,E2 33289.24} C_VEL
LIN {X 0,Y 696.317,Z 1129.236,A -85,B 0,C 180,E1 33287.563,E2 33287.563} C_VEL
LIN {X 0,Y 696.561,Z 1116.859,A -85,B 0,C 180,E1 33285.962,E2 33285.962} C_VEL
LIN {X 0,Y 696.875,Z 1103.057,A -85,B 0,C 180,E1 33284.438,E2 33284.438} C_VEL
LIN {X 0,Y 697.252,Z 1087.753,A -85,B 0,C 180,E1 33282.992,E2 33282.992} C_VEL
LIN {X 0,Y 697.708,Z 1070.832,A -85,B 0,C 180,E1 33281.624,E2 33281.624} C_VEL
LIN {X 0,Y 698.238,Z 1052.171,A -85,B 0,C 180,E1 33280.337,E2 33280.337} C_VEL
LIN {X 0,Y 698.775,Z 1033.04,A -85,B 0,C 180,E1 33279.217,E2 33279.217} C_VEL
LIN {X 0,Y 698.921,Z 1027.536,A -85,B 0,C 180,E1 33278.928,E2 33278.928} C_VEL
LIN {X 0,Y 698.156,Z 1021.129,A -85,B 0,C 180,E1 33278.572,E2 33278.572} C_VEL
LIN {X 0,Y 692.938,Z 1005.126,A -85,B 0,C 180,E1 33277.664,E2 33277.664} C_VEL
LIN {X 0,Y 692.194,Z 998.324,A -85,B 0,C 180,E1 33277.363,E2 33277.363} C_VEL
LIN {X 0,Y 692.747,Z 977.223,A -85,B 0,C 180,E1 33276.616,E2 33276.616} C_VEL
LIN {X 0,Y 693.212,Z 955.65,A -85,B 0,C 180,E1 33276.024,E2 33276.024} C_VEL
LIN {X 0,Y 693.546,Z 933.682,A -85,B 0,C 180,E1 33275.578,E2 33275.578} C_VEL
LIN {X 0,Y 693.827,Z 908.513,A -85,B 0,C 180,E1 33275.242,E2 33275.242} C_VEL
LIN {X 0,Y 695.32,Z 638.086,A -85,B 0,C 180,E1 33272.25,E2 33272.25} C_VEL
LIN {X 0,Y 692.385,Z 627.604,A -85,B 0,C 180,E1 33272.002,E2 33272.002} C_VEL
LIN {X 0,Y 690.817,Z 623.978,A -85,B 0,C 180,E1 33271.872,E2 33271.872} C_VEL
LIN {X 0,Y 688.443,Z 614.914,A -85,B 0,C 180,E1 33270.865,E2 33270.865} C_VEL
LIN {X 0,Y 688.386,Z 614.919,A -85,B 0,C 180,E1 33267.868,E2 33267.868} C_VEL
LIN {X 0,Y 688.411,Z 614.918,A -85,B 0,C 180,E1 33265.15,E2 33265.15} C_VEL
LIN {X 0,Y 688.429,Z 614.909,A -85,B 0,C 180,E1 33262.062,E2 33262.062} C_VEL
LIN {X 0,Y 688.464,Z 614.913,A -85,B 0,C 180,E1 33259.172,E2 33259.172} C_VEL
LIN {X 0,Y 688.462,Z 614.907,A -85,B 0,C 180,E1 33256.085,E2 33256.085} C_VEL
LIN {X 0,Y 688.41,Z 614.913,A -85,B 0,C 180,E1 33253.166,E2 33253.166} C_VEL
LIN {X 0,Y 688.416,Z 614.914,A -85,B 0,C 180,E1 33250.444,E2 33250.444} C_VEL
LIN {X 0,Y 688.391,Z 614.914,A -85,B 0,C 180,E1 33247.395,E2 33247.395} C_VEL
LIN {X 0,Y 688.437,Z 614.914,A -85,B 0,C 180,E1 33244.705,E2 33244.705} C_VEL
LIN {X 0,Y 688.447,Z 614.907,A -85,B 0,C 180,E1 33241.623,E2 33241.623} C_VEL
LIN {X 0,Y 688.442,Z 614.913,A -85,B 0,C 180,E1 33238.64,E2 33238.64} C_VEL
LIN {X 0,Y 688.465,Z 614.907,A -85,B 0,C 180,E1 33235.646,E2 33235.646} C_VEL
LIN {X 0,Y 688.383,Z 614.914,A -85,B 0,C 180,E1 33232.73,E2 33232.73} C_VEL
LIN {X 0,Y 688.412,Z 614.916,A -85,B 0,C 180,E1 33230.047,E2 33230.047} C_VEL
LIN {X 0,Y 688.422,Z 614.909,A -85,B 0,C 180,E1 33227.062,E2 33227.062} C_VEL
LIN {X 0,Y 688.467,Z 614.911,A -85,B 0,C 180,E1 33224.123,E2 33224.123} C_VEL
LIN {X 0,Y 688.456,Z 614.907,A -85,B 0,C 180,E1 33221.054,E2 33221.054} C_VEL
LIN {X 0,Y 688.42,Z 614.911,A -85,B 0,C 180,E1 33218.184,E2 33218.184} C_VEL
LIN {X 0,Y 688.427,Z 614.912,A -85,B 0,C 180,E1 33215.418,E2 33215.418} C_VEL
LIN {X 0,Y 688.383,Z 614.912,A -85,B 0,C 180,E1 33212.415,E2 33212.415} C_VEL
LIN {X 0,Y 688.421,Z 614.914,A -85,B 0,C 180,E1 33209.751,E2 33209.751} C_VEL
LIN {X 0,Y 688.445,Z 614.904,A -85,B 0,C 180,E1 33206.671,E2 33206.671} C_VEL
LIN {X 0,Y 688.449,Z 614.913,A -85,B 0,C 180,E1 33203.664,E2 33203.664} C_VEL
LIN {X 0,Y 688.465,Z 614.906,A -85,B 0,C 180,E1 33200.64,E2 33200.64} C_VEL
LIN {X 0,Y 688.396,Z 614.912,A -85,B 0,C 180,E1 33197.758,E2 33197.758} C_VEL
LIN {X 0,Y 688.389,Z 614.915,A -85,B 0,C 180,E1 33195.19,E2 33195.19} C_VEL
LIN {X 0,Y 688.414,Z 614.911,A -85,B 0,C 180,E1 33192.046,E2 33192.046} C_VEL
LIN {X 0,Y 688.46,Z 614.914,A -85,B 0,C 180,E1 33189.157,E2 33189.157} C_VEL
LIN {X 0,Y 688.454,Z 614.906,A -85,B 0,C 180,E1 33186.097,E2 33186.097} C_VEL
LIN {X 0,Y 688.427,Z 614.912,A -85,B 0,C 180,E1 33183.149,E2 33183.149} C_VEL
LIN {X 0,Y 688.45,Z 614.91,A -85,B 0,C 180,E1 33180.281,E2 33180.281} C_VEL
LIN {X 0,Y 688.378,Z 614.916,A -85,B 0,C 180,E1 33177.295,E2 33177.295} C_VEL
LIN {X 0,Y 688.418,Z 614.915,A -85,B 0,C 180,E1 33174.687,E2 33174.687} C_VEL
LIN {X 0,Y 688.439,Z 614.908,A -85,B 0,C 180,E1 33171.651,E2 33171.651} C_VEL
LIN {X 0,Y 688.459,Z 614.913,A -85,B 0,C 180,E1 33168.662,E2 33168.662} C_VEL
LIN {X 0,Y 688.464,Z 614.908,A -85,B 0,C 180,E1 33165.603,E2 33165.603} C_VEL
LIN {X 0,Y 688.403,Z 614.915,A -85,B 0,C 180,E1 33162.699,E2 33162.699} C_VEL
LIN {X 0,Y 688.401,Z 614.918,A -85,B 0,C 180,E1 33160.046,E2 33160.046} C_VEL
LIN {X 0,Y 688.378,Z 614.941,A -85,B 0,C 180,E1 33158.578,E2 33158.578} C_VEL
LIN {X 0,Y 690.998,Z 625.379,A -85,B 0,C 180,E1 33157.738,E2 33157.738} C_VEL
LIN {X 0,Y 690.745,Z 670.792,A -85,B 0,C 180,E1 33154.468,E2 33154.468} C_VEL
LIN {X 0,Y 690.438,Z 710.904,A -85,B 0,C 180,E1 33151.566,E2 33151.566} C_VEL
LIN {X 0,Y 690.06,Z 751.972,A -85,B 0,C 180,E1 33148.592,E2 33148.592} C_VEL
LIN {X 0,Y 689.554,Z 792.595,A -85,B 0,C 180,E1 33145.645,E2 33145.645} C_VEL
LIN {X 0,Y 689.347,Z 817.738,A -85,B 0,C 180,E1 33143.842,E2 33143.842} C_VEL
LIN {X 0,Y 689.762,Z 826.029,A -85,B 0,C 180,E1 33143.743,E2 33143.743} C_VEL
LIN {X 0,Y 689.363,Z 959.093,A -85,B 0,C 180,E1 33142.315,E2 33142.315} C_VEL
LIN {X 0,Y 689.253,Z 975.475,A -85,B 0,C 180,E1 33141.98,E2 33141.98} C_VEL
LIN {X 0,Y 689.083,Z 992.543,A -85,B 0,C 180,E1 33141.446,E2 33141.446} C_VEL
LIN {X 0,Y 688.902,Z 1005.993,A -85,B 0,C 180,E1 33140.872,E2 33140.872} C_VEL
LIN {X 0,Y 688.746,Z 1018.292,A -85,B 0,C 180,E1 33140.211,E2 33140.211} C_VEL
LIN {X 0,Y 688.582,Z 1028.987,A -85,B 0,C 180,E1 33139.508,E2 33139.508} C_VEL
LIN {X 0,Y 688.418,Z 1039.479,A -85,B 0,C 180,E1 33138.677,E2 33138.677} C_VEL
LIN {X 0,Y 688.266,Z 1049.861,A -85,B 0,C 180,E1 33137.673,E2 33137.673} C_VEL
LIN {X 0,Y 688.129,Z 1059.742,A -85,B 0,C 180,E1 33136.458,E2 33136.458} C_VEL
LIN {X 0,Y 688.05,Z 1066.841,A -85,B 0,C 180,E1 33135.334,E2 33135.334} C_VEL
LIN {X 0,Y 688.007,Z 1072.284,A -85,B 0,C 180,E1 33134.228,E2 33134.228} C_VEL
LIN {X 0,Y 687.974,Z 1076.41,A -85,B 0,C 180,E1 33133.102,E2 33133.102} C_VEL
LIN {X 0,Y 687.96,Z 1079.364,A -85,B 0,C 180,E1 33131.908,E2 33131.908} C_VEL
LIN {X 0,Y 687.952,Z 1081.121,A -85,B 0,C 180,E1 33130.465,E2 33130.465} C_VEL
LIN {X 0,Y 687.958,Z 1080.863,A -85,B 0,C 180,E1 33129.113,E2 33129.113} C_VEL
LIN {X 0,Y 687.965,Z 1079.259,A -85,B 0,C 180,E1 33127.934,E2 33127.934} C_VEL
LIN {X 0,Y 687.981,Z 1076.575,A -85,B 0,C 180,E1 33126.843,E2 33126.843} C_VEL
LIN {X 0,Y 688.011,Z 1072.667,A -85,B 0,C 180,E1 33125.753,E2 33125.753} C_VEL
LIN {X 0,Y 688.053,Z 1067.44,A -85,B 0,C 180,E1 33124.666,E2 33124.666} C_VEL
LIN {X 0,Y 688.131,Z 1060.746,A -85,B 0,C 180,E1 33123.58,E2 33123.58} C_VEL
LIN {X 0,Y 688.257,Z 1051.623,A -85,B 0,C 180,E1 33122.413,E2 33122.413} C_VEL
LIN {X 0,Y 688.429,Z 1040.795,A -85,B 0,C 180,E1 33121.33,E2 33121.33} C_VEL
LIN {X 0,Y 688.597,Z 1029.971,A -85,B 0,C 180,E1 33120.456,E2 33120.456} C_VEL
LIN {X 0,Y 688.766,Z 1017.984,A -85,B 0,C 180,E1 33119.665,E2 33119.665} C_VEL
LIN {X 0,Y 688.928,Z 1004.629,A -85,B 0,C 180,E1 33118.959,E2 33118.959} C_VEL
LIN {X 0,Y 689.122,Z 990.265,A -85,B 0,C 180,E1 33118.377,E2 33118.377} C_VEL
LIN {X 0,Y 689.258,Z 975.694,A -85,B 0,C 180,E1 33117.941,E2 33117.941} C_VEL
LIN {X 0,Y 689.355,Z 960.638,A -85,B 0,C 180,E1 33117.621,E2 33117.621} C_VEL
LIN {X 0,Y 689.455,Z 915.707,A -85,B 0,C 180,E1 33117.121,E2 33117.121} C_VEL
LIN {X 0,Y 689.555,Z 819.313,A -85,B 0,C 180,E1 33116.09,E2 33116.09} C_VEL
LIN {X 0,Y 689.443,Z 817.994,A -85,B 0,C 180,E1 33116.052,E2 33116.052} C_VEL
LIN {X 0,Y 689.903,Z 775.882,A -85,B 0,C 180,E1 33113.006,E2 33113.006} C_VEL
LIN {X 0,Y 690.151,Z 737.72,A -85,B 0,C 180,E1 33110.281,E2 33110.281} C_VEL
LIN {X 0,Y 690.361,Z 700.571,A -85,B 0,C 180,E1 33107.672,E2 33107.672} C_VEL
LIN {X 0,Y 690.225,Z 660.093,A -85,B 0,C 180,E1 33104.884,E2 33104.884} C_VEL
LIN {X 0,Y 690.049,Z 621.634,A -85,B 0,C 180,E1 33102.326,E2 33102.326} C_VEL
LIN {X 0,Y 688.462,Z 614.913,A -85,B 0,C 180,E1 33101.83,E2 33101.83} C_VEL
LIN {X 0,Y 688.438,Z 614.916,A -85,B 0,C 180,E1 33098.797,E2 33098.797} C_VEL
LIN {X 0,Y 688.462,Z 614.917,A -85,B 0,C 180,E1 33095.821,E2 33095.821} C_VEL
LIN {X 0,Y 688.454,Z 614.915,A -85,B 0,C 180,E1 33092.866,E2 33092.866} C_VEL
LIN {X 0,Y 688.468,Z 614.91,A -85,B 0,C 180,E1 33089.781,E2 33089.781} C_VEL
LIN {X 0,Y 688.418,Z 614.915,A -85,B 0,C 180,E1 33086.699,E2 33086.699} C_VEL
LIN {X 0,Y 688.438,Z 614.913,A -85,B 0,C 180,E1 33083.853,E2 33083.853} C_VEL
LIN {X 0,Y 688.453,Z 614.913,A -85,B 0,C 180,E1 33080.817,E2 33080.817} C_VEL
LIN {X 0,Y 688.454,Z 614.915,A -85,B 0,C 180,E1 33077.855,E2 33077.855} C_VEL
LIN {X 0,Y 688.451,Z 614.913,A -85,B 0,C 180,E1 33074.865,E2 33074.865} C_VEL
LIN {X 0,Y 688.446,Z 614.914,A -85,B 0,C 180,E1 33071.918,E2 33071.918} C_VEL
LIN {X 0,Y 688.453,Z 614.911,A -85,B 0,C 180,E1 33068.858,E2 33068.858} C_VEL
LIN {X 0,Y 688.418,Z 614.917,A -85,B 0,C 180,E1 33065.927,E2 33065.927} C_VEL
LIN {X 0,Y 688.468,Z 615.064,A -85,B 0,C 180,E1 33063.595,E2 33063.595} C_VEL
LIN {X 0,Y 693.611,Z 632.247,A -85,B 0,C 180,E1 33061.94,E2 33061.94} C_VEL
LIN {X 0,Y 692.789,Z 667.735,A -85,B 0,C 180,E1 33059.168,E2 33059.168} C_VEL
LIN {X 0,Y 692.579,Z 683.325,A -85,B 0,C 180,E1 33057.994,E2 33057.994} C_VEL
LIN {X 0,Y 695.289,Z 696.911,A -85,B 0,C 180,E1 33057.72,E2 33057.72} C_VEL
LIN {X 0,Y 693.747,Z 977.829,A -85,B 0,C 180,E1 33054.605,E2 33054.605} C_VEL
LIN {X 0,Y 693.499,Z 999.477,A -85,B 0,C 180,E1 33054.278,E2 33054.278} C_VEL
LIN {X 0,Y 693.078,Z 1021.068,A -85,B 0,C 180,E1 33053.795,E2 33053.795} C_VEL
LIN {X 0,Y 692.61,Z 1042.486,A -85,B 0,C 180,E1 33053.164,E2 33053.164} C_VEL
LIN {X 0,Y 692.089,Z 1062.685,A -85,B 0,C 180,E1 33052.42,E2 33052.42} C_VEL
LIN {X 0,Y 691.521,Z 1081.985,A -85,B 0,C 180,E1 33051.545,E2 33051.545} C_VEL
LIN {X 0,Y 690.891,Z 1102.202,A -85,B 0,C 180,E1 33050.456,E2 33050.456} C_VEL
LIN {X 0,Y 690.32,Z 1120.045,A -85,B 0,C 180,E1 33049.325,E2 33049.325} C_VEL
LIN {X 0,Y 689.777,Z 1137.526,A -85,B 0,C 180,E1 33048.022,E2 33048.022} C_VEL
LIN {X 0,Y 689.305,Z 1152.877,A -85,B 0,C 180,E1 33046.69,E2 33046.69} C_VEL
LIN {X 0,Y 688.901,Z 1167.473,A -85,B 0,C 180,E1 33045.229,E2 33045.229} C_VEL
LIN {X 0,Y 688.566,Z 1180.673,A -85,B 0,C 180,E1 33043.69,E2 33043.69} C_VEL
LIN {X 0,Y 688.31,Z 1192.396,A -85,B 0,C 180,E1 33042.073,E2 33042.073} C_VEL
LIN {X 0,Y 688.127,Z 1203.222,A -85,B 0,C 180,E1 33040.294,E2 33040.294} C_VEL
LIN {X 0,Y 688.024,Z 1211.703,A -85,B 0,C 180,E1 33038.608,E2 33038.608} C_VEL
LIN {X 0,Y 687.943,Z 1218.676,A -85,B 0,C 180,E1 33036.844,E2 33036.844} C_VEL
LIN {X 0,Y 687.91,Z 1224.199,A -85,B 0,C 180,E1 33035.002,E2 33035.002} C_VEL
LIN {X 0,Y 687.902,Z 1227.881,A -85,B 0,C 180,E1 33033.249,E2 33033.249} C_VEL
LIN {X 0,Y 687.9,Z 1229.885,A -85,B 0,C 180,E1 33031.498,E2 33031.498} C_VEL
LIN {X 0,Y 687.899,Z 1230.396,A -85,B 0,C 180,E1 33029.582,E2 33029.582} C_VEL
LIN {X 0,Y 687.913,Z 1229.231,A -85,B 0,C 180,E1 33027.75,E2 33027.75} C_VEL
LIN {X 0,Y 687.922,Z 1226.301,A -85,B 0,C 180,E1 33025.915,E2 33025.915} C_VEL
LIN {X 0,Y 687.926,Z 1221.651,A -85,B 0,C 180,E1 33024.076,E2 33024.076} C_VEL
LIN {X 0,Y 687.97,Z 1215.58,A -85,B 0,C 180,E1 33022.315,E2 33022.315} C_VEL
LIN {X 0,Y 688.055,Z 1208.063,A -85,B 0,C 180,E1 33020.632,E2 33020.632} C_VEL
LIN {X 0,Y 688.199,Z 1198.318,A -85,B 0,C 180,E1 33018.857,E2 33018.857} C_VEL
LIN {X 0,Y 688.415,Z 1187.715,A -85,B 0,C 180,E1 33017.245,E2 33017.245} C_VEL
LIN {X 0,Y 688.681,Z 1175.743,A -85,B 0,C 180,E1 33015.71,E2 33015.71} C_VEL
LIN {X 0,Y 689.05,Z 1161.7,A -85,B 0,C 180,E1 33014.168,E2 33014.168} C_VEL
LIN {X 0,Y 689.508,Z 1146.187,A -85,B 0,C 180,E1 33012.705,E2 33012.705} C_VEL
LIN {X 0,Y 690.008,Z 1130.014,A -85,B 0,C 180,E1 33011.392,E2 33011.392} C_VEL
LIN {X 0,Y 690.556,Z 1112.749,A -85,B 0,C 180,E1 33010.194,E2 33010.194} C_VEL
LIN {X 0,Y 691.186,Z 1092.914,A -85,B 0,C 180,E1 33009.019,E2 33009.019} C_VEL
LIN {X 0,Y 691.764,Z 1073.713,A -85,B 0,C 180,E1 33008.059,E2 33008.059} C_VEL
LIN {X 0,Y 692.336,Z 1053.606,A -85,B 0,C 180,E1 33007.228,E2 33007.228} C_VEL
LIN {X 0,Y 692.823,Z 1032.646,A -85,B 0,C 180,E1 33006.526,E2 33006.526} C_VEL
LIN {X 0,Y 693.296,Z 1011.053,A -85,B 0,C 180,E1 33005.961,E2 33005.961} C_VEL
LIN {X 0,Y 693.621,Z 989.77,A -85,B 0,C 180,E1 33005.557,E2 33005.557} C_VEL
LIN {X 0,Y 693.895,Z 956.162,A -85,B 0,C 180,E1 33005.152,E2 33005.152} C_VEL
LIN {X 0,Y 695.25,Z 695.632,A -85,B 0,C 180,E1 33002.264,E2 33002.264} C_VEL
LIN {X 0,Y 692.498,Z 682.766,A -85,B 0,C 180,E1 33001.989,E2 33001.989} C_VEL
LIN {X 0,Y 693.068,Z 643.753,A -85,B 0,C 180,E1 32999.047,E2 32999.047} C_VEL
LIN {X 0,Y 693.093,Z 630.509,A -85,B 0,C 180,E1 32998.026,E2 32998.026} C_VEL
LIN {X 0,Y 688.453,Z 614.916,A -85,B 0,C 180,E1 32996.577,E2 32996.577} C_VEL
LIN {X 0,Y 688.433,Z 614.914,A -85,B 0,C 180,E1 32993.659,E2 32993.659} C_VEL
LIN {X 0,Y 688.459,Z 614.91,A -85,B 0,C 180,E1 32990.711,E2 32990.711} C_VEL
LIN {X 0,Y 688.432,Z 614.915,A -85,B 0,C 180,E1 32987.741,E2 32987.741} C_VEL
LIN {X 0,Y 688.458,Z 614.908,A -85,B 0,C 180,E1 32984.782,E2 32984.782} C_VEL
LIN {X 0,Y 688.428,Z 614.916,A -85,B 0,C 180,E1 32981.7,E2 32981.7} C_VEL
LIN {X 0,Y 688.431,Z 614.91,A -85,B 0,C 180,E1 32978.863,E2 32978.863} C_VEL
LIN {X 0,Y 688.431,Z 614.916,A -85,B 0,C 180,E1 32975.717,E2 32975.717} C_VEL
LIN {X 0,Y 688.406,Z 614.915,A -85,B 0,C 180,E1 32973.004,E2 32973.004} C_VEL
LIN {X 0,Y 688.469,Z 614.914,A -85,B 0,C 180,E1 32970.049,E2 32970.049} C_VEL
LIN {X 0,Y 688.408,Z 615.018,A -85,B 0,C 180,E1 32969.093,E2 32969.093} C_VEL
LIN {X 0,Y 691.078,Z 624.794,A -85,B 0,C 180,E1 32968,E2 32968} C_VEL
LIN {X 0,Y 693.572,Z 631.198,A -85,B 0,C 180,E1 32967.815,E2 32967.815} C_VEL
LIN {X 0,Y 695.276,Z 638.981,A -85,B 0,C 180,E1 32967.652,E2 32967.652} C_VEL
LIN {X 0,Y 693.869,Z 901.462,A -85,B 0,C 180,E1 32964.745,E2 32964.745} C_VEL
LIN {X 0,Y 693.596,Z 931.265,A -85,B 0,C 180,E1 32964.373,E2 32964.373} C_VEL
LIN {X 0,Y 693.279,Z 953.227,A -85,B 0,C 180,E1 32963.947,E2 32963.947} C_VEL
LIN {X 0,Y 692.786,Z 974.558,A -85,B 0,C 180,E1 32963.374,E2 32963.374} C_VEL
LIN {X 0,Y 692.26,Z 995.971,A -85,B 0,C 180,E1 32962.636,E2 32962.636} C_VEL
LIN {X 0,Y 691.685,Z 1016.489,A -85,B 0,C 180,E1 32961.766,E2 32961.766} C_VEL
LIN {X 0,Y 691.088,Z 1036.156,A -85,B 0,C 180,E1 32960.763,E2 32960.763} C_VEL
LIN {X 0,Y 690.488,Z 1055.132,A -85,B 0,C 180,E1 32959.609,E2 32959.609} C_VEL
LIN {X 0,Y 689.906,Z 1073.134,A -85,B 0,C 180,E1 32958.322,E2 32958.322} C_VEL
LIN {X 0,Y 689.395,Z 1089.568,A -85,B 0,C 180,E1 32956.951,E2 32956.951} C_VEL
LIN {X 0,Y 688.978,Z 1104.655,A -85,B 0,C 180,E1 32955.489,E2 32955.489} C_VEL
LIN {X 0,Y 688.633,Z 1118.202,A -85,B 0,C 180,E1 32953.949,E2 32953.949} C_VEL
LIN {X 0,Y 688.352,Z 1130.927,A -85,B 0,C 180,E1 32952.246,E2 32952.246} C_VEL
LIN {X 0,Y 688.157,Z 1141.559,A -85,B 0,C 180,E1 32950.551,E2 32950.551} C_VEL
LIN {X 0,Y 688.036,Z 1150.293,A -85,B 0,C 180,E1 32948.863,E2 32948.863} C_VEL
LIN {X 0,Y 687.964,Z 1157.606,A -85,B 0,C 180,E1 32947.098,E2 32947.098} C_VEL
LIN {X 0,Y 687.934,Z 1163.452,A -85,B 0,C 180,E1 32945.256,E2 32945.256} C_VEL
LIN {X 0,Y 687.918,Z 1167.331,A -85,B 0,C 180,E1 32943.502,E2 32943.502} C_VEL
LIN {X 0,Y 687.913,Z 1169.713,A -85,B 0,C 180,E1 32941.668,E2 32941.668} C_VEL
LIN {X 0,Y 687.91,Z 1170.474,A -85,B 0,C 180,E1 32939.835,E2 32939.835} C_VEL
LIN {X 0,Y 687.91,Z 1169.583,A -85,B 0,C 180,E1 32938.086,E2 32938.086} C_VEL
LIN {X 0,Y 687.912,Z 1167.038,A -85,B 0,C 180,E1 32936.252,E2 32936.252} C_VEL
LIN {X 0,Y 687.928,Z 1162.821,A -85,B 0,C 180,E1 32934.413,E2 32934.413} C_VEL
LIN {X 0,Y 687.973,Z 1157.025,A -85,B 0,C 180,E1 32932.654,E2 32932.654} C_VEL
LIN {X 0,Y 688.054,Z 1149.122,A -85,B 0,C 180,E1 32930.804,E2 32930.804} C_VEL
LIN {X 0,Y 688.18,Z 1140.18,A -85,B 0,C 180,E1 32929.114,E2 32929.114} C_VEL
LIN {X 0,Y 688.376,Z 1129.23,A -85,B 0,C 180,E1 32927.418,E2 32927.418} C_VEL
LIN {X 0,Y 688.657,Z 1116.855,A -85,B 0,C 180,E1 32925.798,E2 32925.798} C_VEL
LIN {X 0,Y 689.024,Z 1103.056,A -85,B 0,C 180,E1 32924.257,E2 32924.257} C_VEL
LIN {X 0,Y 689.457,Z 1087.742,A -85,B 0,C 180,E1 32922.794,E2 32922.794} C_VEL
LIN {X 0,Y 689.955,Z 1071.387,A -85,B 0,C 180,E1 32921.454,E2 32921.454} C_VEL
LIN {X 0,Y 690.536,Z 1053.519,A -85,B 0,C 180,E1 32920.197,E2 32920.197} C_VEL
LIN {X 0,Y 691.137,Z 1034.642,A -85,B 0,C 180,E1 32919.065,E2 32919.065} C_VEL
LIN {X 0,Y 691.751,Z 1014.305,A -85,B 0,C 180,E1 32918.04,E2 32918.04} C_VEL
LIN {X 0,Y 692.194,Z 998.324,A -85,B 0,C 180,E1 32917.363,E2 32917.363} C_VEL
LIN {X 0,Y 691.581,Z 991.423,A -85,B 0,C 180,E1 32917.071,E2 32917.071} C_VEL
LIN {X 0,Y 686.431,Z 974.337,A -85,B 0,C 180,E1 32916.299,E2 32916.299} C_VEL
LIN {X 0,Y 685.616,Z 967.226,A -85,B 0,C 180,E1 32916.053,E2 32916.053} C_VEL
LIN {X 0,Y 686.044,Z 945.686,A -85,B 0,C 180,E1 32915.528,E2 32915.528} C_VEL
LIN {X 0,Y 686.427,Z 922.734,A -85,B 0,C 180,E1 32915.135,E2 32915.135} C_VEL
LIN {X 0,Y 688.13,Z 652.856,A -85,B 0,C 180,E1 32912.109,E2 32912.109} C_VEL
LIN {X 0,Y 688.011,Z 638.834,A -85,B 0,C 180,E1 32911.94,E2 32911.94} C_VEL
LIN {X 0,Y 685.867,Z 631.236,A -85,B 0,C 180,E1 32911.752,E2 32911.752} C_VEL
LIN {X 0,Y 682.671,Z 624.151,A -85,B 0,C 180,E1 32911.499,E2 32911.499} C_VEL
LIN {X 0,Y 680.531,Z 615.902,A -85,B 0,C 180,E1 32910.57,E2 32910.57} C_VEL
LIN {X 0,Y 680.439,Z 615.909,A -85,B 0,C 180,E1 32907.666,E2 32907.666} C_VEL
LIN {X 0,Y 680.52,Z 615.903,A -85,B 0,C 180,E1 32904.779,E2 32904.779} C_VEL
LIN {X 0,Y 680.481,Z 615.9,A -85,B 0,C 180,E1 32901.788,E2 32901.788} C_VEL
LIN {X 0,Y 680.513,Z 615.899,A -85,B 0,C 180,E1 32898.918,E2 32898.918} C_VEL
LIN {X 0,Y 680.521,Z 615.899,A -85,B 0,C 180,E1 32895.861,E2 32895.861} C_VEL
LIN {X 0,Y 680.466,Z 615.902,A -85,B 0,C 180,E1 32892.969,E2 32892.969} C_VEL
LIN {X 0,Y 680.526,Z 615.902,A -85,B 0,C 180,E1 32890.053,E2 32890.053} C_VEL
LIN {X 0,Y 680.45,Z 615.903,A -85,B 0,C 180,E1 32887.154,E2 32887.154} C_VEL
LIN {X 0,Y 680.525,Z 615.902,A -85,B 0,C 180,E1 32884.341,E2 32884.341} C_VEL
LIN {X 0,Y 680.5,Z 615.898,A -85,B 0,C 180,E1 32881.343,E2 32881.343} C_VEL
LIN {X 0,Y 680.496,Z 615.9,A -85,B 0,C 180,E1 32878.43,E2 32878.43} C_VEL
LIN {X 0,Y 680.528,Z 615.9,A -85,B 0,C 180,E1 32875.407,E2 32875.407} C_VEL
LIN {X 0,Y 680.44,Z 615.903,A -85,B 0,C 180,E1 32872.554,E2 32872.554} C_VEL
LIN {X 0,Y 680.525,Z 615.902,A -85,B 0,C 180,E1 32869.65,E2 32869.65} C_VEL
LIN {X 0,Y 680.474,Z 615.9,A -85,B 0,C 180,E1 32866.739,E2 32866.739} C_VEL
LIN {X 0,Y 680.516,Z 615.896,A -85,B 0,C 180,E1 32863.858,E2 32863.858} C_VEL
LIN {X 0,Y 680.516,Z 615.899,A -85,B 0,C 180,E1 32860.841,E2 32860.841} C_VEL
LIN {X 0,Y 680.475,Z 615.898,A -85,B 0,C 180,E1 32857.94,E2 32857.94} C_VEL
LIN {X 0,Y 680.522,Z 615.904,A -85,B 0,C 180,E1 32854.974,E2 32854.974} C_VEL
LIN {X 0,Y 680.439,Z 615.901,A -85,B 0,C 180,E1 32852.106,E2 32852.106} C_VEL
LIN {X 0,Y 680.528,Z 615.902,A -85,B 0,C 180,E1 32849.328,E2 32849.328} C_VEL
LIN {X 0,Y 680.494,Z 615.895,A -85,B 0,C 180,E1 32846.294,E2 32846.294} C_VEL
LIN {X 0,Y 680.501,Z 615.899,A -85,B 0,C 180,E1 32843.42,E2 32843.42} C_VEL
LIN {X 0,Y 680.526,Z 615.898,A -85,B 0,C 180,E1 32840.444,E2 32840.444} C_VEL
LIN {X 0,Y 680.452,Z 615.9,A -85,B 0,C 180,E1 32837.613,E2 32837.613} C_VEL
LIN {X 0,Y 680.491,Z 615.904,A -85,B 0,C 180,E1 32834.84,E2 32834.84} C_VEL
LIN {X 0,Y 680.468,Z 615.9,A -85,B 0,C 180,E1 32831.851,E2 32831.851} C_VEL
LIN {X 0,Y 680.525,Z 615.902,A -85,B 0,C 180,E1 32828.993,E2 32828.993} C_VEL
LIN {X 0,Y 680.512,Z 615.896,A -85,B 0,C 180,E1 32825.985,E2 32825.985} C_VEL
LIN {X 0,Y 680.488,Z 615.901,A -85,B 0,C 180,E1 32823.093,E2 32823.093} C_VEL
LIN {X 0,Y 680.53,Z 615.899,A -85,B 0,C 180,E1 32820.128,E2 32820.128} C_VEL
LIN {X 0,Y 680.437,Z 615.905,A -85,B 0,C 180,E1 32817.192,E2 32817.192} C_VEL
LIN {X 0,Y 680.51,Z 615.905,A -85,B 0,C 180,E1 32814.421,E2 32814.421} C_VEL
LIN {X 0,Y 680.49,Z 615.899,A -85,B 0,C 180,E1 32811.412,E2 32811.412} C_VEL
LIN {X 0,Y 680.51,Z 615.901,A -85,B 0,C 180,E1 32808.499,E2 32808.499} C_VEL
LIN {X 0,Y 680.524,Z 615.899,A -85,B 0,C 180,E1 32805.444,E2 32805.444} C_VEL
LIN {X 0,Y 680.461,Z 615.904,A -85,B 0,C 180,E1 32802.595,E2 32802.595} C_VEL
LIN {X 0,Y 680.487,Z 615.906,A -85,B 0,C 180,E1 32799.837,E2 32799.837} C_VEL
LIN {X 0,Y 680.444,Z 615.944,A -85,B 0,C 180,E1 32798.796,E2 32798.796} C_VEL
LIN {X 0,Y 683.372,Z 627.362,A -85,B 0,C 180,E1 32797.862,E2 32797.862} C_VEL
LIN {X 0,Y 683.077,Z 671.718,A -85,B 0,C 180,E1 32794.652,E2 32794.652} C_VEL
LIN {X 0,Y 682.756,Z 710.81,A -85,B 0,C 180,E1 32791.815,E2 32791.815} C_VEL
LIN {X 0,Y 682.348,Z 751.963,A -85,B 0,C 180,E1 32788.82,E2 32788.82} C_VEL
LIN {X 0,Y 681.794,Z 793.612,A -85,B 0,C 180,E1 32785.785,E2 32785.785} C_VEL
LIN {X 0,Y 681.591,Z 818.577,A -85,B 0,C 180,E1 32783.995,E2 32783.995} C_VEL
LIN {X 0,Y 681.992,Z 826.798,A -85,B 0,C 180,E1 32783.895,E2 32783.895} C_VEL
LIN {X 0,Y 681.536,Z 960.058,A -85,B 0,C 180,E1 32782.441,E2 32782.441} C_VEL
LIN {X 0,Y 681.422,Z 976.401,A -85,B 0,C 180,E1 32782.101,E2 32782.101} C_VEL
LIN {X 0,Y 681.252,Z 993.264,A -85,B 0,C 180,E1 32781.569,E2 32781.569} C_VEL
LIN {X 0,Y 681.05,Z 1007.568,A -85,B 0,C 180,E1 32780.949,E2 32780.949} C_VEL
LIN {X 0,Y 680.871,Z 1020.723,A -85,B 0,C 180,E1 32780.221,E2 32780.221} C_VEL
LIN {X 0,Y 680.674,Z 1032.874,A -85,B 0,C 180,E1 32779.387,E2 32779.387} C_VEL
LIN {X 0,Y 680.467,Z 1045.171,A -85,B 0,C 180,E1 32778.326,E2 32778.326} C_VEL
LIN {X 0,Y 680.299,Z 1054.876,A -85,B 0,C 180,E1 32777.269,E2 32777.269} C_VEL
LIN {X 0,Y 680.185,Z 1062.695,A -85,B 0,C 180,E1 32776.216,E2 32776.216} C_VEL
LIN {X 0,Y 680.108,Z 1069.407,A -85,B 0,C 180,E1 32775.081,E2 32775.081} C_VEL
LIN {X 0,Y 680.055,Z 1075.235,A -85,B 0,C 180,E1 32773.778,E2 32773.778} C_VEL
LIN {X 0,Y 680.025,Z 1079.529,A -85,B 0,C 180,E1 32772.308,E2 32772.308} C_VEL
LIN {X 0,Y 680.013,Z 1081.501,A -85,B 0,C 180,E1 32771.104,E2 32771.104} C_VEL
LIN {X 0,Y 680.013,Z 1082.133,A -85,B 0,C 180,E1 32769.819,E2 32769.819} C_VEL
LIN {X 0,Y 680.016,Z 1081.045,A -85,B 0,C 180,E1 32768.368,E2 32768.368} C_VEL
LIN {X 0,Y 680.049,Z 1077.901,A -85,B 0,C 180,E1 32766.923,E2 32766.923} C_VEL
LIN {X 0,Y 680.091,Z 1073.409,A -85,B 0,C 180,E1 32765.651,E2 32765.651} C_VEL
LIN {X 0,Y 680.151,Z 1067.656,A -85,B 0,C 180,E1 32764.467,E2 32764.467} C_VEL
LIN {X 0,Y 680.253,Z 1059.523,A -85,B 0,C 180,E1 32763.2,E2 32763.2} C_VEL
LIN {X 0,Y 680.407,Z 1050.482,A -85,B 0,C 180,E1 32762.104,E2 32762.104} C_VEL
LIN {X 0,Y 680.584,Z 1040.075,A -85,B 0,C 180,E1 32761.093,E2 32761.093} C_VEL
LIN {X 0,Y 680.792,Z 1028.314,A -85,B 0,C 180,E1 32760.166,E2 32760.166} C_VEL
LIN {X 0,Y 680.967,Z 1014.906,A -85,B 0,C 180,E1 32759.325,E2 32759.325} C_VEL
LIN {X 0,Y 681.171,Z 1000.302,A -85,B 0,C 180,E1 32758.61,E2 32758.61} C_VEL
LIN {X 0,Y 681.337,Z 986.503,A -85,B 0,C 180,E1 32758.106,E2 32758.106} C_VEL
LIN {X 0,Y 681.437,Z 974.47,A -85,B 0,C 180,E1 32757.767,E2 32757.767} C_VEL
LIN {X 0,Y 681.523,Z 960.496,A -85,B 0,C 180,E1 32757.481,E2 32757.481} C_VEL
LIN {X 0,Y 681.792,Z 820.043,A -85,B 0,C 180,E1 32755.937,E2 32755.937} C_VEL
LIN {X 0,Y 681.738,Z 818.2,A -85,B 0,C 180,E1 32755.835,E2 32755.835} C_VEL
LIN {X 0,Y 682.189,Z 775.039,A -85,B 0,C 180,E1 32752.715,E2 32752.715} C_VEL
LIN {X 0,Y 682.437,Z 740.076,A -85,B 0,C 180,E1 32750.213,E2 32750.213} C_VEL
LIN {X 0,Y 682.666,Z 701.827,A -85,B 0,C 180,E1 32747.522,E2 32747.522} C_VEL
LIN {X 0,Y 682.541,Z 663.403,A -85,B 0,C 180,E1 32744.877,E2 32744.877} C_VEL
LIN {X 0,Y 682.437,Z 624.144,A -85,B 0,C 180,E1 32742.255,E2 32742.255} C_VEL
LIN {X 0,Y 680.523,Z 615.903,A -85,B 0,C 180,E1 32741.646,E2 32741.646} C_VEL
LIN {X 0,Y 680.525,Z 615.904,A -85,B 0,C 180,E1 32738.538,E2 32738.538} C_VEL
LIN {X 0,Y 680.503,Z 615.907,A -85,B 0,C 180,E1 32735.52,E2 32735.52} C_VEL
LIN {X 0,Y 680.495,Z 615.904,A -85,B 0,C 180,E1 32732.617,E2 32732.617} C_VEL
LIN {X 0,Y 680.52,Z 615.899,A -85,B 0,C 180,E1 32729.443,E2 32729.443} C_VEL
LIN {X 0,Y 680.488,Z 615.904,A -85,B 0,C 180,E1 32726.461,E2 32726.461} C_VEL
LIN {X 0,Y 680.523,Z 615.902,A -85,B 0,C 180,E1 32723.481,E2 32723.481} C_VEL
LIN {X 0,Y 680.524,Z 615.902,A -85,B 0,C 180,E1 32720.475,E2 32720.475} C_VEL
LIN {X 0,Y 680.526,Z 615.899,A -85,B 0,C 180,E1 32717.362,E2 32717.362} C_VEL
LIN {X 0,Y 680.48,Z 615.903,A -85,B 0,C 180,E1 32714.307,E2 32714.307} C_VEL
LIN {X 0,Y 680.514,Z 615.901,A -85,B 0,C 180,E1 32711.337,E2 32711.337} C_VEL
LIN {X 0,Y 680.512,Z 615.903,A -85,B 0,C 180,E1 32708.313,E2 32708.313} C_VEL
LIN {X 0,Y 680.517,Z 615.905,A -85,B 0,C 180,E1 32705.365,E2 32705.365} C_VEL
LIN {X 0,Y 680.531,Z 615.973,A -85,B 0,C 180,E1 32703.938,E2 32703.938} C_VEL
LIN {X 0,Y 686.226,Z 635.01,A -85,B 0,C 180,E1 32702.078,E2 32702.078} C_VEL
LIN {X 0,Y 685.288,Z 670.737,A -85,B 0,C 180,E1 32699.259,E2 32699.259} C_VEL
LIN {X 0,Y 685.104,Z 683.138,A -85,B 0,C 180,E1 32698.317,E2 32698.317} C_VEL
LIN {X 0,Y 688.166,Z 698.246,A -85,B 0,C 180,E1 32698.01,E2 32698.01} C_VEL
LIN {X 0,Y 686.477,Z 977.528,A -85,B 0,C 180,E1 32694.887,E2 32694.887} C_VEL
LIN {X 0,Y 686.195,Z 999.152,A -85,B 0,C 180,E1 32694.559,E2 32694.559} C_VEL
LIN {X 0,Y 685.737,Z 1020.74,A -85,B 0,C 180,E1 32694.075,E2 32694.075} C_VEL
LIN {X 0,Y 685.189,Z 1042.964,A -85,B 0,C 180,E1 32693.413,E2 32693.413} C_VEL
LIN {X 0,Y 684.597,Z 1063.454,A -85,B 0,C 180,E1 32692.646,E2 32692.646} C_VEL
LIN {X 0,Y 683.959,Z 1082.881,A -85,B 0,C 180,E1 32691.751,E2 32691.751} C_VEL
LIN {X 0,Y 683.276,Z 1102.198,A -85,B 0,C 180,E1 32690.694,E2 32690.694} C_VEL
LIN {X 0,Y 682.644,Z 1120.024,A -85,B 0,C 180,E1 32689.552,E2 32689.552} C_VEL
LIN {X 0,Y 682.03,Z 1137.467,A -85,B 0,C 180,E1 32688.239,E2 32688.239} C_VEL
LIN {X 0,Y 681.493,Z 1152.877,A -85,B 0,C 180,E1 32686.887,E2 32686.887} C_VEL
LIN {X 0,Y 681.034,Z 1167.474,A -85,B 0,C 180,E1 32685.41,E2 32685.41} C_VEL
LIN {X 0,Y 680.656,Z 1180.885,A -85,B 0,C 180,E1 32683.826,E2 32683.826} C_VEL
LIN {X 0,Y 680.372,Z 1192.395,A -85,B 0,C 180,E1 32682.216,E2 32682.216} C_VEL
LIN {X 0,Y 680.164,Z 1203.223,A -85,B 0,C 180,E1 32680.416,E2 32680.416} C_VEL
LIN {X 0,Y 680.038,Z 1211.703,A -85,B 0,C 180,E1 32678.709,E2 32678.709} C_VEL
LIN {X 0,Y 679.951,Z 1218.677,A -85,B 0,C 180,E1 32676.925,E2 32676.925} C_VEL
LIN {X 0,Y 679.913,Z 1224.199,A -85,B 0,C 180,E1 32675.061,E2 32675.061} C_VEL
LIN {X 0,Y 679.905,Z 1227.88,A -85,B 0,C 180,E1 32673.287,E2 32673.287} C_VEL
LIN {X 0,Y 679.901,Z 1229.885,A -85,B 0,C 180,E1 32671.516,E2 32671.516} C_VEL
LIN {X 0,Y 679.899,Z 1230.396,A -85,B 0,C 180,E1 32669.578,E2 32669.578} C_VEL
LIN {X 0,Y 679.913,Z 1229.231,A -85,B 0,C 180,E1 32667.723,E2 32667.723} C_VEL
LIN {X 0,Y 679.923,Z 1226.3,A -85,B 0,C 180,E1 32665.867,E2 32665.867} C_VEL
LIN {X 0,Y 679.932,Z 1221.651,A -85,B 0,C 180,E1 32664.006,E2 32664.006} C_VEL
LIN {X 0,Y 679.982,Z 1215.58,A -85,B 0,C 180,E1 32662.224,E2 32662.224} C_VEL
LIN {X 0,Y 680.077,Z 1208.063,A -85,B 0,C 180,E1 32660.521,E2 32660.521} C_VEL
LIN {X 0,Y 680.244,Z 1198.317,A -85,B 0,C 180,E1 32658.725,E2 32658.725} C_VEL
LIN {X 0,Y 680.49,Z 1187.714,A -85,B 0,C 180,E1 32657.094,E2 32657.094} C_VEL
LIN {X 0,Y 680.789,Z 1175.745,A -85,B 0,C 180,E1 32655.54,E2 32655.54} C_VEL
LIN {X 0,Y 681.208,Z 1161.699,A -85,B 0,C 180,E1 32653.98,E2 32653.98} C_VEL
LIN {X 0,Y 681.728,Z 1146.187,A -85,B 0,C 180,E1 32652.501,E2 32652.501} C_VEL
LIN {X 0,Y 682.308,Z 1129.672,A -85,B 0,C 180,E1 32651.147,E2 32651.147} C_VEL
LIN {X 0,Y 682.916,Z 1112.236,A -85,B 0,C 180,E1 32649.929,E2 32649.929} C_VEL
LIN {X 0,Y 683.61,Z 1092.91,A -85,B 0,C 180,E1 32648.776,E2 32648.776} C_VEL
LIN {X 0,Y 684.262,Z 1073.708,A -85,B 0,C 180,E1 32647.805,E2 32647.805} C_VEL
LIN {X 0,Y 684.895,Z 1053.603,A -85,B 0,C 180,E1 32646.966,E2 32646.966} C_VEL
LIN {X 0,Y 685.45,Z 1032.644,A -85,B 0,C 180,E1 32646.258,E2 32646.258} C_VEL
LIN {X 0,Y 685.965,Z 1011.015,A -85,B 0,C 180,E1 32645.687,E2 32645.687} C_VEL
LIN {X 0,Y 686.338,Z 989.607,A -85,B 0,C 180,E1 32645.278,E2 32645.278} C_VEL
LIN {X 0,Y 686.641,Z 955.239,A -85,B 0,C 180,E1 32644.861,E2 32644.861} C_VEL
LIN {X 0,Y 688.095,Z 697.011,A -85,B 0,C 180,E1 32641.98,E2 32641.98} C_VEL
LIN {X 0,Y 684.928,Z 681.965,A -85,B 0,C 180,E1 32641.654,E2 32641.654} C_VEL
LIN {X 0,Y 685.595,Z 643.133,A -85,B 0,C 180,E1 32638.69,E2 32638.69} C_VEL
LIN {X 0,Y 685.66,Z 633.252,A -85,B 0,C 180,E1 32637.917,E2 32637.917} C_VEL
LIN {X 0,Y 680.521,Z 615.904,A -85,B 0,C 180,E1 32636.261,E2 32636.261} C_VEL
LIN {X 0,Y 680.508,Z 615.899,A -85,B 0,C 180,E1 32633.206,E2 32633.206} C_VEL
LIN {X 0,Y 680.517,Z 615.903,A -85,B 0,C 180,E1 32630.052,E2 32630.052} C_VEL
LIN {X 0,Y 680.504,Z 615.898,A -85,B 0,C 180,E1 32627.017,E2 32627.017} C_VEL
LIN {X 0,Y 680.5,Z 615.905,A -85,B 0,C 180,E1 32623.825,E2 32623.825} C_VEL
LIN {X 0,Y 680.492,Z 615.899,A -85,B 0,C 180,E1 32620.946,E2 32620.946} C_VEL
LIN {X 0,Y 680.495,Z 615.905,A -85,B 0,C 180,E1 32617.766,E2 32617.766} C_VEL
LIN {X 0,Y 680.475,Z 615.902,A -85,B 0,C 180,E1 32614.966,E2 32614.966} C_VEL
LIN {X 0,Y 680.52,Z 615.904,A -85,B 0,C 180,E1 32611.936,E2 32611.936} C_VEL
LIN {X 0,Y 680.482,Z 616.012,A -85,B 0,C 180,E1 32609.45,E2 32609.45} C_VEL
LIN {X 0,Y 683.248,Z 625.592,A -85,B 0,C 180,E1 32608.348,E2 32608.348} C_VEL
LIN {X 0,Y 686.797,Z 633.966,A -85,B 0,C 180,E1 32608.083,E2 32608.083} C_VEL
LIN {X 0,Y 688.159,Z 640.434,A -85,B 0,C 180,E1 32607.942,E2 32607.942} C_VEL
LIN {X 0,Y 686.6,Z 902.403,A -85,B 0,C 180,E1 32605.014,E2 32605.014} C_VEL
LIN {X 0,Y 686.296,Z 931.693,A -85,B 0,C 180,E1 32604.642,E2 32604.642} C_VEL
LIN {X 0,Y 685.936,Z 953.575,A -85,B 0,C 180,E1 32604.211,E2 32604.211} C_VEL
LIN {X 0,Y 685.393,Z 975.005,A -85,B 0,C 180,E1 32603.628,E2 32603.628} C_VEL
LIN {X 0,Y 684.815,Z 995.983,A -85,B 0,C 180,E1 32602.896,E2 32602.896} C_VEL
LIN {X 0,Y 684.163,Z 1016.493,A -85,B 0,C 180,E1 32602.018,E2 32602.018} C_VEL
LIN {X 0,Y 683.507,Z 1036.171,A -85,B 0,C 180,E1 32601.004,E2 32601.004} C_VEL
LIN {X 0,Y 682.84,Z 1054.79,A -85,B 0,C 180,E1 32599.861,E2 32599.861} C_VEL
LIN {X 0,Y 682.175,Z 1073.008,A -85,B 0,C 180,E1 32598.547,E2 32598.547} C_VEL
LIN {X 0,Y 681.599,Z 1089.57,A -85,B 0,C 180,E1 32597.151,E2 32597.151} C_VEL
LIN {X 0,Y 681.124,Z 1104.657,A -85,B 0,C 180,E1 32595.672,E2 32595.672} C_VEL
LIN {X 0,Y 680.732,Z 1118.209,A -85,B 0,C 180,E1 32594.114,E2 32594.114} C_VEL
LIN {X 0,Y 680.42,Z 1130.344,A -85,B 0,C 180,E1 32592.477,E2 32592.477} C_VEL
LIN {X 0,Y 680.2,Z 1141.092,A -85,B 0,C 180,E1 32590.761,E2 32590.761} C_VEL
LIN {X 0,Y 680.062,Z 1149.891,A -85,B 0,C 180,E1 32589.053,E2 32589.053} C_VEL
LIN {X 0,Y 679.976,Z 1157.606,A -85,B 0,C 180,E1 32587.182,E2 32587.182} C_VEL
LIN {X 0,Y 679.937,Z 1163.452,A -85,B 0,C 180,E1 32585.318,E2 32585.318} C_VEL
LIN {X 0,Y 679.917,Z 1167.333,A -85,B 0,C 180,E1 32583.543,E2 32583.543} C_VEL
LIN {X 0,Y 679.913,Z 1169.712,A -85,B 0,C 180,E1 32581.687,E2 32581.687} C_VEL
LIN {X 0,Y 679.909,Z 1170.474,A -85,B 0,C 180,E1 32579.833,E2 32579.833} C_VEL
LIN {X 0,Y 679.909,Z 1169.582,A -85,B 0,C 180,E1 32578.064,E2 32578.064} C_VEL
LIN {X 0,Y 679.91,Z 1167.038,A -85,B 0,C 180,E1 32576.207,E2 32576.207} C_VEL
LIN {X 0,Y 679.931,Z 1163.055,A -85,B 0,C 180,E1 32574.432,E2 32574.432} C_VEL
LIN {X 0,Y 679.979,Z 1157.33,A -85,B 0,C 180,E1 32572.652,E2 32572.652} C_VEL
LIN {X 0,Y 680.069,Z 1149.527,A -85,B 0,C 180,E1 32570.78,E2 32570.78} C_VEL
LIN {X 0,Y 680.21,Z 1140.667,A -85,B 0,C 180,E1 32569.071,E2 32569.071} C_VEL
LIN {X 0,Y 680.428,Z 1129.809,A -85,B 0,C 180,E1 32567.354,E2 32567.354} C_VEL
LIN {X 0,Y 680.759,Z 1116.847,A -85,B 0,C 180,E1 32565.63,E2 32565.63} C_VEL
LIN {X 0,Y 681.186,Z 1102.761,A -85,B 0,C 180,E1 32564.04,E2 32564.04} C_VEL
LIN {X 0,Y 681.672,Z 1087.731,A -85,B 0,C 180,E1 32562.591,E2 32562.591} C_VEL
LIN {X 0,Y 682.237,Z 1071.214,A -85,B 0,C 180,E1 32561.224,E2 32561.224} C_VEL
LIN {X 0,Y 682.889,Z 1053.07,A -85,B 0,C 180,E1 32559.937,E2 32559.937} C_VEL
LIN {X 0,Y 683.588,Z 1033.836,A -85,B 0,C 180,E1 32558.778,E2 32558.778} C_VEL
LIN {X 0,Y 684.264,Z 1013.812,A -85,B 0,C 180,E1 32557.764,E2 32557.764} C_VEL
LIN {X 0,Y 684.894,Z 993.538,A -85,B 0,C 180,E1 32556.92,E2 32556.92} C_VEL
LIN {X 0,Y 685.476,Z 971.999,A -85,B 0,C 180,E1 32556.193,E2 32556.193} C_VEL
LIN {X 0,Y 685.616,Z 967.226,A -85,B 0,C 180,E1 32556.053,E2 32556.053} C_VEL
LIN {X 0,Y 684.898,Z 960.015,A -85,B 0,C 180,E1 32555.819,E2 32555.819} C_VEL
LIN {X 0,Y 679.766,Z 942.001,A -85,B 0,C 180,E1 32555.205,E2 32555.205} C_VEL
LIN {X 0,Y 678.953,Z 934.57,A -85,B 0,C 180,E1 32555.034,E2 32555.034} C_VEL
LIN {X 0,Y 679.291,Z 911.173,A -85,B 0,C 180,E1 32554.707,E2 32554.707} C_VEL
LIN {X 0,Y 681.114,Z 644.099,A -85,B 0,C 180,E1 32551.696,E2 32551.696} C_VEL
LIN {X 0,Y 680.836,Z 639.983,A -85,B 0,C 180,E1 32551.632,E2 32551.632} C_VEL
LIN {X 0,Y 679.046,Z 634.167,A -85,B 0,C 180,E1 32551.477,E2 32551.477} C_VEL
LIN {X 0,Y 674.656,Z 624.678,A -85,B 0,C 180,E1 32551.153,E2 32551.153} C_VEL
LIN {X 0,Y 672.572,Z 616.894,A -85,B 0,C 180,E1 32550.252,E2 32550.252} C_VEL
LIN {X 0,Y 672.5,Z 616.898,A -85,B 0,C 180,E1 32547.462,E2 32547.462} C_VEL
LIN {X 0,Y 672.578,Z 616.89,A -85,B 0,C 180,E1 32544.462,E2 32544.462} C_VEL
LIN {X 0,Y 672.547,Z 616.89,A -85,B 0,C 180,E1 32541.581,E2 32541.581} C_VEL
LIN {X 0,Y 672.578,Z 616.884,A -85,B 0,C 180,E1 32538.585,E2 32538.585} C_VEL
LIN {X 0,Y 672.574,Z 616.892,A -85,B 0,C 180,E1 32535.44,E2 32535.44} C_VEL
LIN {X 0,Y 672.542,Z 616.889,A -85,B 0,C 180,E1 32532.569,E2 32532.569} C_VEL
LIN {X 0,Y 672.507,Z 616.894,A -85,B 0,C 180,E1 32529.411,E2 32529.411} C_VEL
LIN {X 0,Y 672.535,Z 616.893,A -85,B 0,C 180,E1 32526.704,E2 32526.704} C_VEL
LIN {X 0,Y 672.558,Z 616.886,A -85,B 0,C 180,E1 32523.577,E2 32523.577} C_VEL
LIN {X 0,Y 672.578,Z 616.89,A -85,B 0,C 180,E1 32520.602,E2 32520.602} C_VEL
LIN {X 0,Y 672.585,Z 616.887,A -85,B 0,C 180,E1 32517.539,E2 32517.539} C_VEL
LIN {X 0,Y 672.525,Z 616.892,A -85,B 0,C 180,E1 32514.602,E2 32514.602} C_VEL
LIN {X 0,Y 672.549,Z 616.892,A -85,B 0,C 180,E1 32511.82,E2 32511.82} C_VEL
LIN {X 0,Y 672.517,Z 616.89,A -85,B 0,C 180,E1 32508.823,E2 32508.823} C_VEL
LIN {X 0,Y 672.586,Z 616.892,A -85,B 0,C 180,E1 32505.965,E2 32505.965} C_VEL
LIN {X 0,Y 672.566,Z 616.884,A -85,B 0,C 180,E1 32502.886,E2 32502.886} C_VEL
LIN {X 0,Y 672.552,Z 616.887,A -85,B 0,C 180,E1 32499.932,E2 32499.932} C_VEL
LIN {X 0,Y 672.591,Z 616.888,A -85,B 0,C 180,E1 32496.917,E2 32496.917} C_VEL
LIN {X 0,Y 672.498,Z 616.892,A -85,B 0,C 180,E1 32494.094,E2 32494.094} C_VEL
LIN {X 0,Y 672.589,Z 616.889,A -85,B 0,C 180,E1 32491.109,E2 32491.109} C_VEL
LIN {X 0,Y 672.541,Z 616.889,A -85,B 0,C 180,E1 32488.127,E2 32488.127} C_VEL
LIN {X 0,Y 672.576,Z 616.882,A -85,B 0,C 180,E1 32485.14,E2 32485.14} C_VEL
LIN {X 0,Y 672.586,Z 616.893,A -85,B 0,C 180,E1 32482.054,E2 32482.054} C_VEL
LIN {X 0,Y 672.541,Z 616.883,A -85,B 0,C 180,E1 32479.118,E2 32479.118} C_VEL
LIN {X 0,Y 672.513,Z 616.893,A -85,B 0,C 180,E1 32475.976,E2 32475.976} C_VEL
LIN {X 0,Y 672.52,Z 616.892,A -85,B 0,C 180,E1 32473.326,E2 32473.326} C_VEL
LIN {X 0,Y 672.56,Z 616.885,A -85,B 0,C 180,E1 32470.188,E2 32470.188} C_VEL
LIN {X 0,Y 672.584,Z 616.891,A -85,B 0,C 180,E1 32467.171,E2 32467.171} C_VEL
LIN {X 0,Y 672.585,Z 616.885,A -85,B 0,C 180,E1 32464.075,E2 32464.075} C_VEL
LIN {X 0,Y 672.529,Z 616.891,A -85,B 0,C 180,E1 32461.107,E2 32461.107} C_VEL
LIN {X 0,Y 672.564,Z 616.892,A -85,B 0,C 180,E1 32458.247,E2 32458.247} C_VEL
LIN {X 0,Y 672.512,Z 616.892,A -85,B 0,C 180,E1 32455.291,E2 32455.291} C_VEL
LIN {X 0,Y 672.585,Z 616.892,A -85,B 0,C 180,E1 32452.447,E2 32452.447} C_VEL
LIN {X 0,Y 672.564,Z 616.887,A -85,B 0,C 180,E1 32449.373,E2 32449.373} C_VEL
LIN {X 0,Y 672.558,Z 616.889,A -85,B 0,C 180,E1 32446.504,E2 32446.504} C_VEL
LIN {X 0,Y 672.591,Z 616.89,A -85,B 0,C 180,E1 32443.493,E2 32443.493} C_VEL
LIN {X 0,Y 672.502,Z 616.897,A -85,B 0,C 180,E1 32440.631,E2 32440.631} C_VEL
LIN {X 0,Y 672.513,Z 616.906,A -85,B 0,C 180,E1 32439.021,E2 32439.021} C_VEL
LIN {X 0,Y 675.757,Z 630.021,A -85,B 0,C 180,E1 32437.943,E2 32437.943} C_VEL
LIN {X 0,Y 675.404,Z 673.802,A -85,B 0,C 180,E1 32434.754,E2 32434.754} C_VEL
LIN {X 0,Y 675.048,Z 714.088,A -85,B 0,C 180,E1 32431.821,E2 32431.821} C_VEL
LIN {X 0,Y 674.598,Z 754.815,A -85,B 0,C 180,E1 32428.843,E2 32428.843} C_VEL
LIN {X 0,Y 674.033,Z 795.707,A -85,B 0,C 180,E1 32425.855,E2 32425.855} C_VEL
LIN {X 0,Y 673.83,Z 819.338,A -85,B 0,C 180,E1 32424.152,E2 32424.152} C_VEL
LIN {X 0,Y 674.227,Z 827.348,A -85,B 0,C 180,E1 32424.054,E2 32424.054} C_VEL
LIN {X 0,Y 673.71,Z 960.814,A -85,B 0,C 180,E1 32422.572,E2 32422.572} C_VEL
LIN {X 0,Y 673.597,Z 976.972,A -85,B 0,C 180,E1 32422.234,E2 32422.234} C_VEL
LIN {X 0,Y 673.439,Z 992.733,A -85,B 0,C 180,E1 32421.741,E2 32421.741} C_VEL
LIN {X 0,Y 673.223,Z 1007.514,A -85,B 0,C 180,E1 32421.108,E2 32421.108} C_VEL
LIN {X 0,Y 673.021,Z 1021.375,A -85,B 0,C 180,E1 32420.341,E2 32420.341} C_VEL
LIN {X 0,Y 672.802,Z 1033.768,A -85,B 0,C 180,E1 32419.481,E2 32419.481} C_VEL
LIN {X 0,Y 672.571,Z 1046.467,A -85,B 0,C 180,E1 32418.369,E2 32418.369} C_VEL
LIN {X 0,Y 672.39,Z 1056.123,A -85,B 0,C 180,E1 32417.3,E2 32417.3} C_VEL
LIN {X 0,Y 672.254,Z 1064.807,A -85,B 0,C 180,E1 32416.095,E2 32416.095} C_VEL
LIN {X 0,Y 672.16,Z 1071.879,A -85,B 0,C 180,E1 32414.822,E2 32414.822} C_VEL
LIN {X 0,Y 672.111,Z 1077.506,A -85,B 0,C 180,E1 32413.417,E2 32413.417} C_VEL
LIN {X 0,Y 672.075,Z 1081.262,A -85,B 0,C 180,E1 32411.933,E2 32411.933} C_VEL
LIN {X 0,Y 672.063,Z 1082.958,A -85,B 0,C 180,E1 32410.542,E2 32410.542} C_VEL
LIN {X 0,Y 672.076,Z 1082.766,A -85,B 0,C 180,E1 32409.072,E2 32409.072} C_VEL
LIN {X 0,Y 672.096,Z 1080.822,A -85,B 0,C 180,E1 32407.693,E2 32407.693} C_VEL
LIN {X 0,Y 672.13,Z 1077.087,A -85,B 0,C 180,E1 32406.318,E2 32406.318} C_VEL
LIN {X 0,Y 672.201,Z 1071.438,A -85,B 0,C 180,E1 32404.947,E2 32404.947} C_VEL
LIN {X 0,Y 672.303,Z 1064.133,A -85,B 0,C 180,E1 32403.665,E2 32403.665} C_VEL
LIN {X 0,Y 672.455,Z 1055.362,A -85,B 0,C 180,E1 32402.47,E2 32402.47} C_VEL
LIN {X 0,Y 672.646,Z 1044.978,A -85,B 0,C 180,E1 32401.361,E2 32401.361} C_VEL
LIN {X 0,Y 672.865,Z 1033.586,A -85,B 0,C 180,E1 32400.381,E2 32400.381} C_VEL
LIN {X 0,Y 673.078,Z 1020.484,A -85,B 0,C 180,E1 32399.487,E2 32399.487} C_VEL
LIN {X 0,Y 673.268,Z 1006.315,A -85,B 0,C 180,E1 32398.722,E2 32398.722} C_VEL
LIN {X 0,Y 673.463,Z 991.684,A -85,B 0,C 180,E1 32398.126,E2 32398.126} C_VEL
